FUNCTION "Automatico_linea_2" : VOID	// FC 6
NAME : Auto_L2
VERSION : 0.1
BEGIN
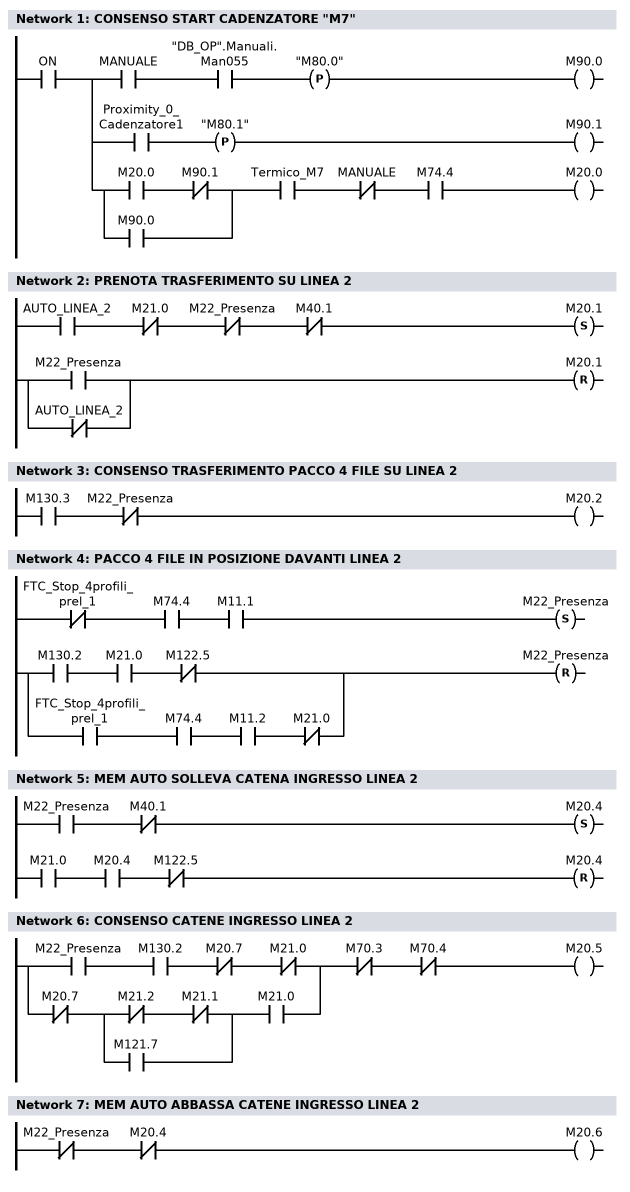
NETWORK
TITLE = CONSENSO START CADENZATORE "M7"
      A     "ON";
      =     L 0.0;
      A     L 0.0;
      A     "MANUALE";
      A     "DB_OP".Manuali.Man055;
      FP    "M80.0";
      =     "M90.0";
      A     L 0.0;
      A     "Proximity_0_Cadenzatore1";
      FP    "M80.1";
      =     "M90.1";
      A     L 0.0;
      A(;
      A     "M20.0";
      AN    "M90.1";
      O     "M90.0";
      );
      A     "Termico_M7";
      AN    "MANUALE";
      A     "M74.4";
      =     "M20.0";
NETWORK
TITLE = PRENOTA TRASFERIMENTO SU LINEA 2
      A     "AUTO_LINEA_2";
      AN    "M21.0";
      AN    "M22_Presenza";
      AN    "M40.1";
      S     "M20.1";
      A(;
      O     "M22_Presenza";
      ON    "AUTO_LINEA_2";
      );
      R     "M20.1";
      NOP   0;
NETWORK
TITLE = CONSENSO TRASFERIMENTO PACCO 4 FILE SU LINEA 2
      A     "M130.3";
      AN    "M22_Presenza";
      =     "M20.2";
NETWORK
TITLE = PACCO 4 FILE IN POSIZIONE DAVANTI LINEA 2
      AN    "FTC_Stop_4profili_prel_1";
      A     "M74.4";
      A     "M11.1";
      S     "M22_Presenza";
      A(;
      A     "M130.2";
      A     "M21.0";
      AN    "M122.5";
      O;
      A     "FTC_Stop_4profili_prel_1";
      A     "M74.4";
      A     "M11.2";
      AN    "M21.0";
      );
      R     "M22_Presenza";
      NOP   0;
NETWORK
TITLE = MEM AUTO SOLLEVA CATENA INGRESSO LINEA 2
      A     "M22_Presenza";
      AN    "M40.1";
      S     "M20.4";
      A     "M21.0";
      A     "M20.4";
      AN    "M122.5";
      R     "M20.4";
      NOP   0;
NETWORK
TITLE = CONSENSO CATENE INGRESSO LINEA 2
      A(;
      A     "M22_Presenza";
      A     "M130.2";
      AN    "M20.7";
      AN    "M21.0";
      O;
      AN    "M20.7";
      A(;
      AN    "M21.2";
      AN    "M21.1";
      O     "M121.7";
      );
      A     "M21.0";
      );
      AN    "M70.3";
      AN    "M70.4";
      =     "M20.5";
NETWORK
TITLE = MEM AUTO ABBASSA CATENE INGRESSO LINEA 2
      AN    "M22_Presenza";
      AN    "M20.4";
      =     "M20.6";
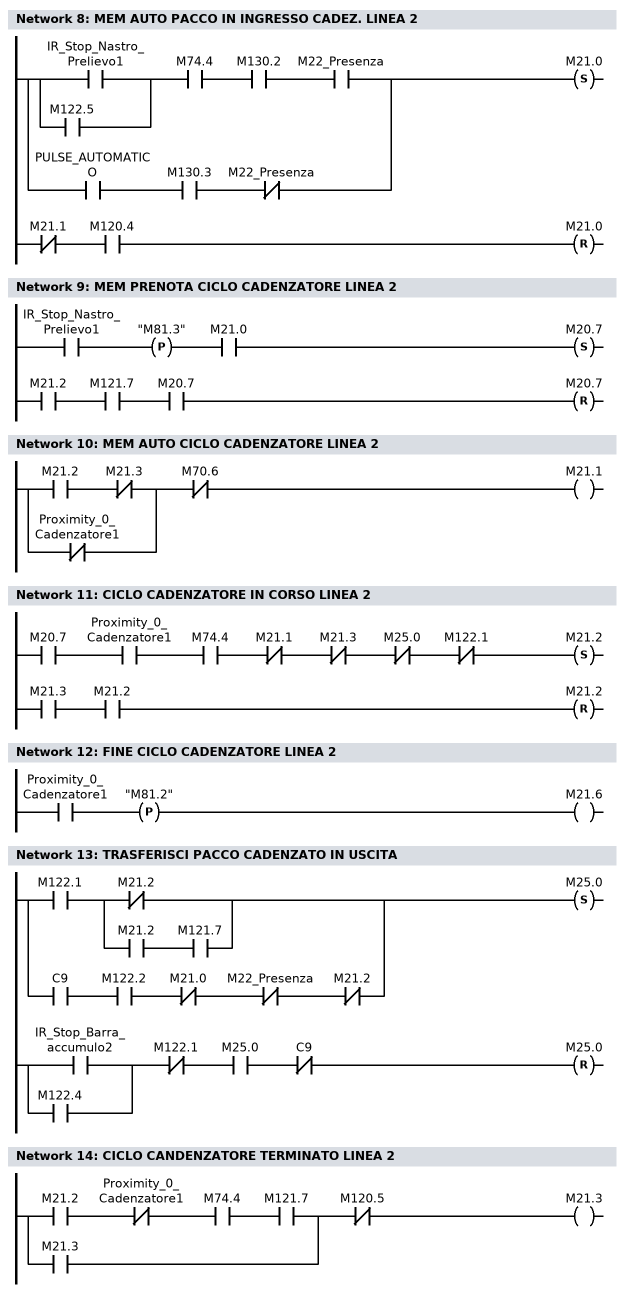
NETWORK
TITLE = MEM AUTO PACCO IN INGRESSO CADEZ. LINEA 2
      A(;
      A(;
      O     "IR_Stop_Nastro_Prelievo1";
      O     "M122.5";
      );
      A     "M74.4";
      A     "M130.2";
      A     "M22_Presenza";
      O;
      A     "PULSE_AUTOMATICO";
      A     "M130.3";
      AN    "M22_Presenza";
      );
      S     "M21.0";
      AN    "M21.1";
      A     "M120.4";
      R     "M21.0";
      NOP   0;
NETWORK
TITLE = MEM PRENOTA CICLO CADENZATORE LINEA 2
      A     "IR_Stop_Nastro_Prelievo1";
      FP    "M81.3";
      A     "M21.0";
      S     "M20.7";
      A     "M21.2";
      A     "M121.7";
      A     "M20.7";
      R     "M20.7";
      NOP   0;
NETWORK
TITLE = MEM AUTO CICLO CADENZATORE LINEA 2
      A(;
      A     "M21.2";
      AN    "M21.3";
      ON    "Proximity_0_Cadenzatore1";
      );
      AN    "M70.6";
      =     "M21.1";
NETWORK
TITLE = CICLO CADENZATORE IN CORSO LINEA 2
      A     "M20.7";
      A     "Proximity_0_Cadenzatore1";
      A     "M74.4";
      AN    "M21.1";
      AN    "M21.3";
      AN    "M25.0";
      AN    "M122.1";
      S     "M21.2";
      A     "M21.3";
      A     "M21.2";
      R     "M21.2";
      NOP   0;
NETWORK
TITLE = FINE CICLO CADENZATORE LINEA 2
      A     "Proximity_0_Cadenzatore1";
      FP    "M81.2";
      =     "M21.6";
NETWORK
TITLE = TRASFERISCI PACCO CADENZATO IN USCITA
      A(;
      A     "M122.1";
      A(;
      ON    "M21.2";
      O;
      A     "M21.2";
      A     "M121.7";
      );
      O;
      A     "C9";
      A     "M122.2";
      AN    "M21.0";
      AN    "M22_Presenza";
      AN    "M21.2";
      );
      S     "M25.0";
      A(;
      O     "IR_Stop_Barra_accumulo2";
      O     "M122.4";
      );
      AN    "M122.1";
      A     "M25.0";
      AN    "C9";
      R     "M25.0";
      NOP   0;
NETWORK
TITLE = CICLO CANDENZATORE TERMINATO LINEA 2
      A(;
      A     "M21.2";
      AN    "Proximity_0_Cadenzatore1";
      A     "M74.4";
      A     "M121.7";
      O     "M21.3";
      );
      AN    "M120.5";
      =     "M21.3";
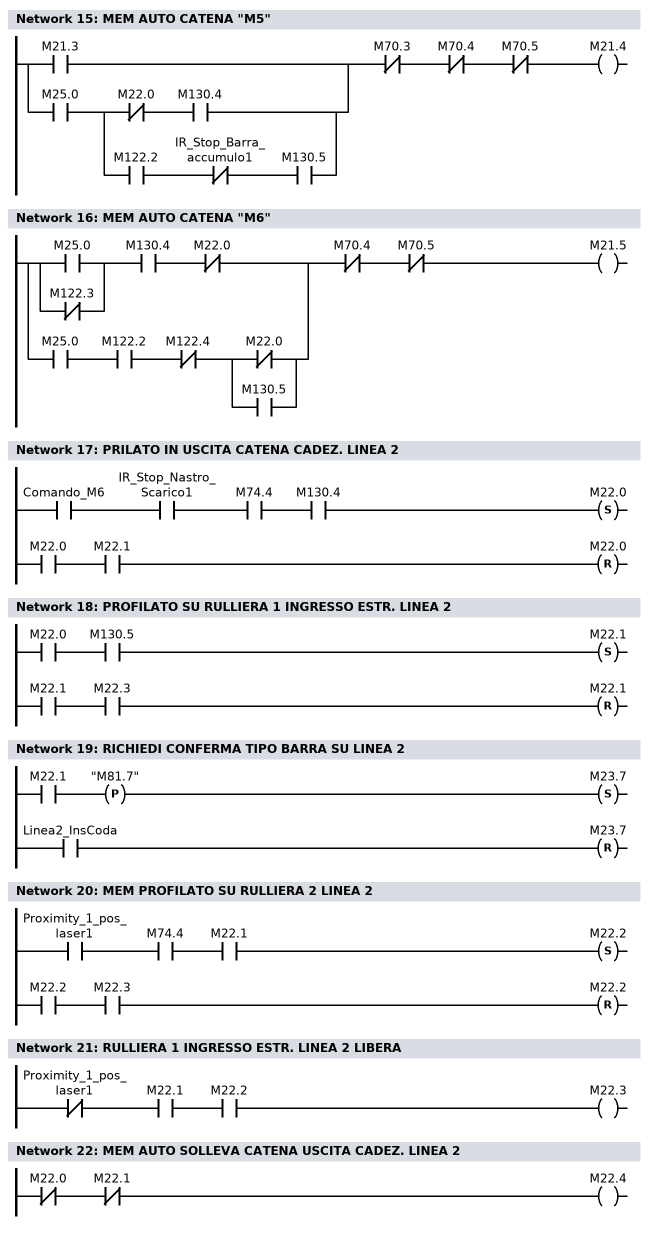
NETWORK
TITLE = MEM AUTO CATENA "M5"
      A(;
      O     "M21.3";
      O;
      A     "M25.0";
      A(;
      AN    "M22.0";
      A     "M130.4";
      O;
      A     "M122.2";
      AN    "IR_Stop_Barra_accumulo1";
      A     "M130.5";
      );
      );
      AN    "M70.3";
      AN    "M70.4";
      AN    "M70.5";
      =     "M21.4";
NETWORK
TITLE = MEM AUTO CATENA "M6"
      A(;
      A(;
      O     "M25.0";
      ON    "M122.3";
      );
      A     "M130.4";
      AN    "M22.0";
      O;
      A     "M25.0";
      A     "M122.2";
      AN    "M122.4";
      A(;
      ON    "M22.0";
      O     "M130.5";
      );
      );
      AN    "M70.4";
      AN    "M70.5";
      =     "M21.5";
NETWORK
TITLE = PRILATO IN USCITA CATENA CADEZ. LINEA 2
      A     "Comando_M6";
      A     "IR_Stop_Nastro_Scarico1";
      A     "M74.4";
      A     "M130.4";
      S     "M22.0";
      A     "M22.0";
      A     "M22.1";
      R     "M22.0";
      NOP   0;
NETWORK
TITLE = PROFILATO SU RULLIERA 1 INGRESSO ESTR. LINEA 2
      A     "M22.0";
      A     "M130.5";
      S     "M22.1";
      A     "M22.1";
      A     "M22.3";
      R     "M22.1";
      NOP   0;
NETWORK
TITLE = RICHIEDI CONFERMA TIPO BARRA SU LINEA 2
      A     "M22.1";
      FP    "M81.7";
      S     "M23.7";
      A     "Linea2_InsCoda";
      R     "M23.7";
      NOP   0;
NETWORK
TITLE = MEM PROFILATO SU RULLIERA 2 LINEA 2
      A     "Proximity_1_pos_laser1";
      A     "M74.4";
      A     "M22.1";
      S     "M22.2";
      A     "M22.2";
      A     "M22.3";
      R     "M22.2";
      NOP   0;
NETWORK
TITLE = RULLIERA 1 INGRESSO ESTR. LINEA 2 LIBERA
      AN    "Proximity_1_pos_laser1";
      A     "M22.1";
      A     "M22.2";
      =     "M22.3";
NETWORK
TITLE = MEM AUTO SOLLEVA CATENA USCITA CADEZ. LINEA 2
      AN    "M22.0";
      AN    "M22.1";
      =     "M22.4";
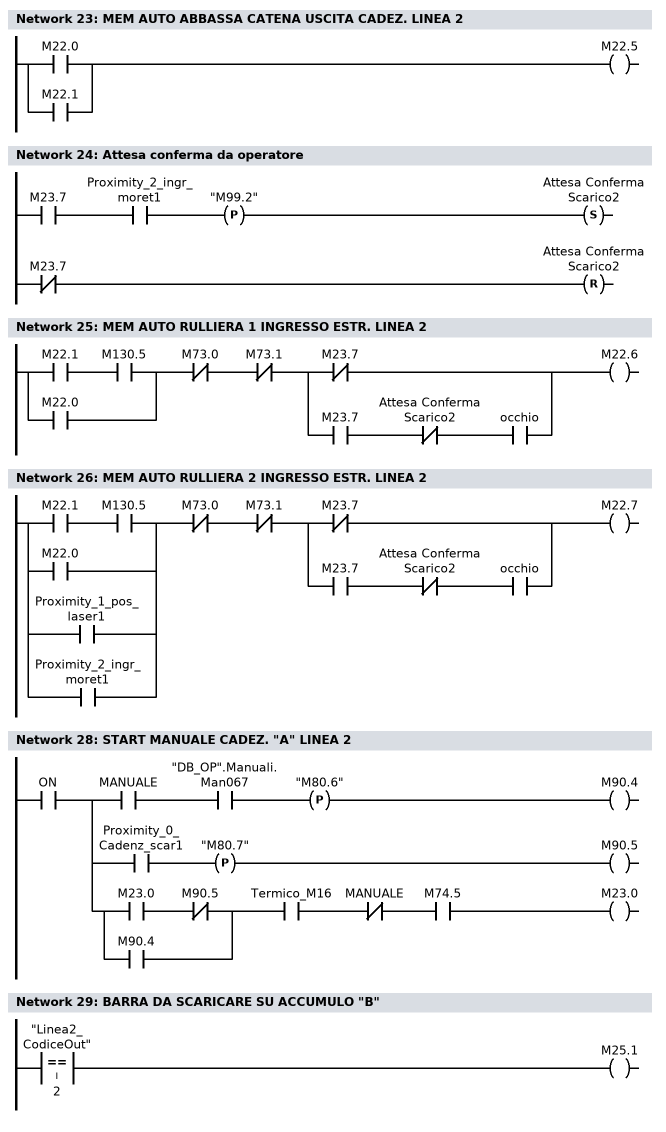
NETWORK
TITLE = MEM AUTO ABBASSA CATENA USCITA CADEZ. LINEA 2
      O     "M22.0";
      O     "M22.1";
      =     "M22.5";
NETWORK
TITLE = Attesa conferma da operatore
      A     "M23.7";
      A     "Proximity_2_ingr_moret1";
      FP    "M99.2";
      S     "Attesa Conferma Scarico2";
      AN    "M23.7";
      R     "Attesa Conferma Scarico2";
      NOP   0;
NETWORK
TITLE = MEM AUTO RULLIERA 1 INGRESSO ESTR. LINEA 2
      A(;
      A     "M22.1";
      A     "M130.5";
      O     "M22.0";
      );
      AN    "M73.0";
      AN    "M73.1";
      A(;
      ON    "M23.7";
      O;
      A     "M23.7";
      AN    "Attesa Conferma Scarico2";
      A     "occhio";
      );
      =     "M22.6";
NETWORK
TITLE = MEM AUTO RULLIERA 2 INGRESSO ESTR. LINEA 2
      A(;
      A     "M22.1";
      A     "M130.5";
      O     "M22.0";
      O     "Proximity_1_pos_laser1";
      O     "Proximity_2_ingr_moret1";
      );
      AN    "M73.0";
      AN    "M73.1";
      A(;
      ON    "M23.7";
      O;
      A     "M23.7";
      AN    "Attesa Conferma Scarico2";
      A     "occhio";
      );
      =     "M22.7";
NETWORK
TITLE =
NETWORK
TITLE = START MANUALE CADEZ. "A" LINEA 2
      A     "ON";
      =     L 0.0;
      A     L 0.0;
      A     "MANUALE";
      A     "DB_OP".Manuali.Man067;
      FP    "M80.6";
      =     "M90.4";
      A     L 0.0;
      A     "Proximity_0_Cadenz_scar1";
      FP    "M80.7";
      =     "M90.5";
      A     L 0.0;
      A(;
      A     "M23.0";
      AN    "M90.5";
      O     "M90.4";
      );
      A     "Termico_M16";
      AN    "MANUALE";
      A     "M74.5";
      =     "M23.0";
NETWORK
TITLE = BARRA DA SCARICARE SU ACCUMULO "B"
      L     "Linea2_CodiceOut";
      L     2;
      ==I;
      =     "M25.1";
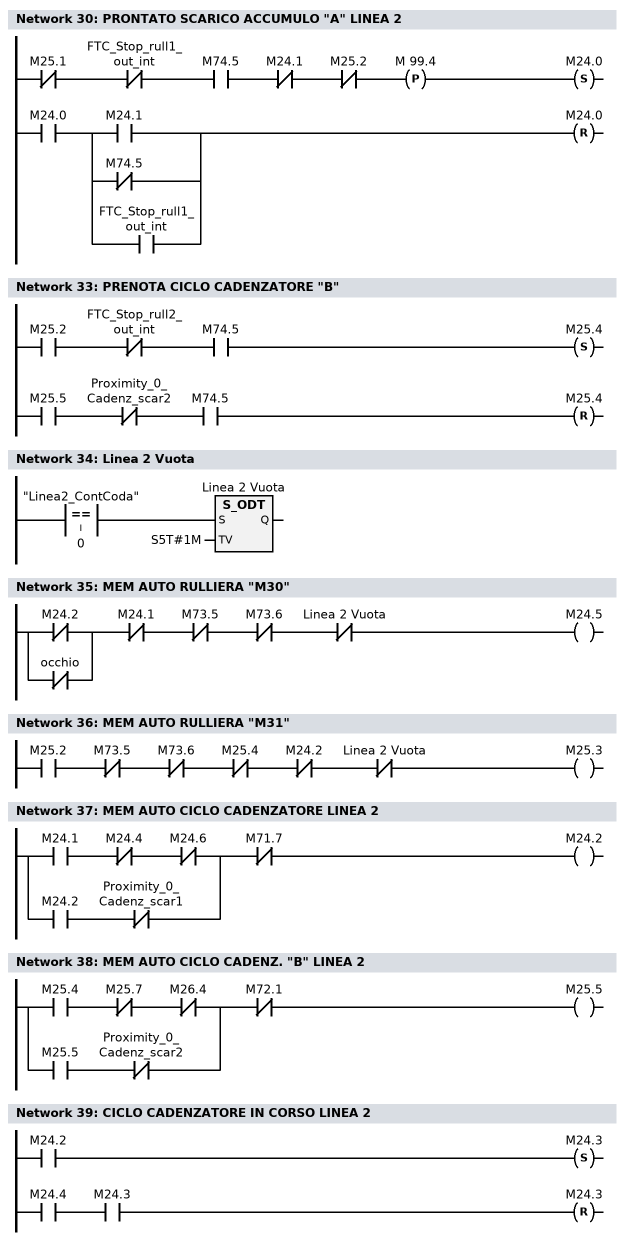
NETWORK
TITLE = PRONTATO SCARICO ACCUMULO "A" LINEA 2
      AN    "M25.1";
      AN    "FTC_Stop_rull1_out_int";
      A     "M74.5";
      AN    "M24.1";
      AN    "M25.2";
      FP    M 99.4;
      S     "M24.0";
      A     "M24.0";
      A(;
      O     "M24.1";
      ON    "M74.5";
      O     "FTC_Stop_rull1_out_int";
      );
      R     "M24.0";
      NOP   0;
NETWORK
TITLE = SPOSTA BASSA RU RULLIERA "M31"
      A(;
      A     "M25.1";
      AN    "FTC_Stop_rull1_out_int";
      A     "M74.5";
      AN    "M24.1";
      S     "M25.2";
      A(;
      A     "M25.4";
      A     "occhio";
      O     "M25.7";
      );
      A     "M25.2";
      R     "M25.2";
      A     "M25.2";
      );
      FP    "M82.1";
      S     "Linea2_DelCoda";
NETWORK
TITLE = PROFILATO PRONTO SU CADEZ. "A" LINEA 2
      A(;
      A(;
      AN    "FTC_Stop_rull1_out_int";
      L     S5T#100MS;
      SD    "T124";
      NOP   0;
      NOP   0;
      NOP   0;
      A     "T124";
      );
      A     "M24.0";
      A     "M74.5";
      S     "M24.1";
      A     "M24.2";
      AN    "Proximity_0_Cadenz_scar1";
      A     "M74.5";
      R     "M24.1";
      A     "M24.1";
      );
      FP    "M82.0";
      S     "Linea2_DelCoda";
NETWORK
TITLE = PRENOTA CICLO CADENZATORE "B"
      A     "M25.2";
      AN    "FTC_Stop_rull2_out_int";
      A     "M74.5";
      S     "M25.4";
      A     "M25.5";
      AN    "Proximity_0_Cadenz_scar2";
      A     "M74.5";
      R     "M25.4";
      NOP   0;
NETWORK
TITLE = Linea 2 Vuota
      A(;
      L     "Linea2_ContCoda";
      L     0;
      ==I;
      );
      L     S5T#1M;
      SD    "Linea 2 Vuota";
      NOP   0;
      NOP   0;
      NOP   0;
      NOP   0;
NETWORK
TITLE = MEM AUTO RULLIERA "M30"
      A(;
      ON    "M24.2";
      ON    "occhio";
      );
      AN    "M24.1";
      AN    "M73.5";
      AN    "M73.6";
      AN    "Linea 2 Vuota";
      =     "M24.5";
NETWORK
TITLE = MEM AUTO RULLIERA "M31"
      A     "M25.2";
      AN    "M73.5";
      AN    "M73.6";
      AN    "M25.4";
      AN    "M24.2";
      AN    "Linea 2 Vuota";
      =     "M25.3";
NETWORK
TITLE = MEM AUTO CICLO CADENZATORE LINEA 2
      A(;
      A     "M24.1";
      AN    "M24.4";
      AN    "M24.6";
      O;
      A     "M24.2";
      AN    "Proximity_0_Cadenz_scar1";
      );
      AN    "M71.7";
      =     "M24.2";
NETWORK
TITLE = MEM AUTO CICLO CADENZ. "B" LINEA 2
      A(;
      A     "M25.4";
      AN    "M25.7";
      AN    "M26.4";
      O;
      A     "M25.5";
      AN    "Proximity_0_Cadenz_scar2";
      );
      AN    "M72.1";
      =     "M25.5";
NETWORK
TITLE = CICLO CADENZATORE IN CORSO LINEA 2
      A     "M24.2";
      S     "M24.3";
      A     "M24.4";
      A     "M24.3";
      R     "M24.3";
      NOP   0;
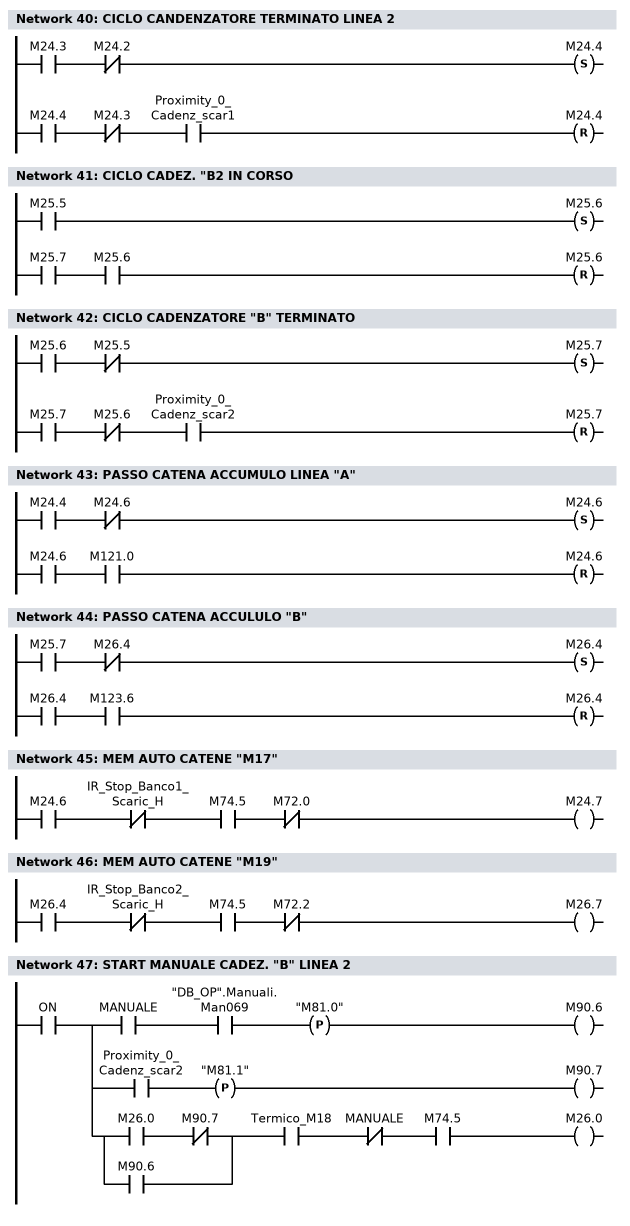
NETWORK
TITLE = CICLO CANDENZATORE TERMINATO LINEA 2
      A     "M24.3";
      AN    "M24.2";
      S     "M24.4";
      A     "M24.4";
      AN    "M24.3";
      A     "Proximity_0_Cadenz_scar1";
      R     "M24.4";
      NOP   0;
NETWORK
TITLE = CICLO CADEZ. "B2 IN CORSO
      A     "M25.5";
      S     "M25.6";
      A     "M25.7";
      A     "M25.6";
      R     "M25.6";
      NOP   0;
NETWORK
TITLE = CICLO CADENZATORE "B" TERMINATO
      A     "M25.6";
      AN    "M25.5";
      S     "M25.7";
      A     "M25.7";
      AN    "M25.6";
      A     "Proximity_0_Cadenz_scar2";
      R     "M25.7";
      NOP   0;
NETWORK
TITLE = PASSO CATENA ACCUMULO LINEA "A"
      A     "M24.4";
      AN    "M24.6";
      S     "M24.6";
      A     "M24.6";
      A     "M121.0";
      R     "M24.6";
      NOP   0;
NETWORK
TITLE = PASSO CATENA ACCULULO "B"
      A     "M25.7";
      AN    "M26.4";
      S     "M26.4";
      A     "M26.4";
      A     "M123.6";
      R     "M26.4";
      NOP   0;
NETWORK
TITLE = MEM AUTO CATENE "M17"
      A     "M24.6";
      AN    "IR_Stop_Banco1_Scaric_H";
      A     "M74.5";
      AN    "M72.0";
      =     "M24.7";
NETWORK
TITLE = MEM AUTO CATENE "M19"
      A     "M26.4";
      AN    "IR_Stop_Banco2_Scaric_H";
      A     "M74.5";
      AN    "M72.2";
      =     "M26.7";
NETWORK
TITLE = START MANUALE CADEZ. "B" LINEA 2
      A     "ON";
      =     L 0.0;
      A     L 0.0;
      A     "MANUALE";
      A     "DB_OP".Manuali.Man069;
      FP    "M81.0";
      =     "M90.6";
      A     L 0.0;
      A     "Proximity_0_Cadenz_scar2";
      FP    "M81.1";
      =     "M90.7";
      A     L 0.0;
      A(;
      A     "M26.0";
      AN    "M90.7";
      O     "M90.6";
      );
      A     "Termico_M18";
      AN    "MANUALE";
      A     "M74.5";
      =     "M26.0";
END_FUNCTION

FUNCTION "PROFIBUS_MM4" : VOID	// FC 10
AUTHOR : PROTEKNO
NAME : MM4
VERSION : 0.1
VAR_INPUT
  Periferic_Address : INT ;
  Drive_On_Off : BOOL ;
  Drive_Reversing : BOOL ;
  Drive_Fault_ACKN : BOOL ;
  Drive_F_Setpoint : REAL ;
END_VAR
VAR_OUTPUT
  Drive_in_operation : BOOL ;
  Drive_Fault_Active : BOOL ;
  Drive_Alarm_Active : BOOL ;
  Freno : BOOL ;
  Drive_F_Act : REAL ;
END_VAR
VAR_TEMP
  Address_E_A : DWORD ;
  SEND : STRUCT
   CW1 : UDT 1;
   f_setpoint : WORD ;
  END_STRUCT ;
  REC : STRUCT
   SW1 : UDT 2;
   f_act : WORD ;
  END_STRUCT ;
END_VAR
BEGIN
NETWORK
TITLE = Trasferimento indirizzo blocco;
      L     #Periferic_Address;
      SLD   3;
      T     #Address_E_A;
NETWORK
TITLE = Status word PZD MM4;
      L     PID [#Address_E_A];
      T     #REC;	//Status word MM4;
NETWORK
TITLE = control bit`s + setpoint
// ---------------------------------------
// IN-Variablen FC
// --------------------------------------
// PZD1 - Steuerwort 1                  // set single bit in the control word 1
      SET;	// set VKE=1
      =     #SEND.CW1.Bit_1;
      =     #SEND.CW1.Bit_2;
      =     #SEND.CW1.Bit_3;
      =     #SEND.CW1.Bit_4;
      =     #SEND.CW1.Bit_5;
      =     #SEND.CW1.Bit_6;
      =     #SEND.CW1.Bit_10;	// setpoint valid
      CLR;	// set VKE=0
      =     #SEND.CW1.Bit_8;
      =     #SEND.CW1.Bit_9;
      =     #SEND.CW1.Bit_12;
      =     #SEND.CW1.Bit_13;
      =     #SEND.CW1.Bit_14;
      =     #SEND.CW1.Bit_15;
      A     #Drive_On_Off;	// on / off ?
      =     #SEND.CW1.Bit_0;
      A     #Drive_Reversing;	// cw / cww ?
      =     #SEND.CW1.Bit_11;
      A     #Drive_Fault_ACKN;	// fault ackn.?
      =     #SEND.CW1.Bit_7;
//  
// PZD2 - Drehzahlsollwert
// gültiger Drehzahlsollwert zwischen 0.00-50 Hz
      L     #Drive_F_Setpoint;	// setpoint [Hz]
      L     0.000000e+00;
      <R;	// setpoinz >0Hz
      JC    N004;
      L     #Drive_F_Setpoint;
      L     7.500000e+01;
      >R;	// setpoint < 75Hz ?
      JC    N004;
      L     #Drive_F_Setpoint;
      L     1.000000e+02;	// 2-Nachkommastellen retten
      *R;
      RND;	//conversion of a 32-bit IEEE floating-point number to 32-bit integer
      L     24576;	// 16384 = 4000HEX = 50Hz
      *D;
      L     7500;
      /D;
      T     #SEND.f_setpoint;
N004: NOP   0;
NETWORK
TITLE = stateword + actual frequency 
// -------------------------------------
// OUT-Variablen FC                     
// -------------------------------------
// PZD 1 - Zustandswort
      A     #REC.SW1.Bit_2;
      =     #Drive_in_operation;
      A     #REC.SW1.Bit_3;
      =     #Drive_Fault_Active;
      A     #REC.SW1.Bit_7;
      =     #Drive_Alarm_Active;
      A     #REC.SW1.Bit_12;
      =     #Freno;
// PZD 2 - Drehzahlistwert
      L     #REC.f_act;
      ITD;
      DTR;
      L     5.000000e+01;	//16383= 4000HEX = 50Hz
      *R;
      L     1.638400e+04;
      /R;
      L     1.000000e+02;
      *R;
      TRUNC;
      ITD;
      DTR;
      L     1.000000e+02;
      /R;
      T     #Drive_F_Act;
NETWORK
TITLE = Control word PZD MM4;
      L     #SEND;	//Control word MM4;
      T     PQD [#Address_E_A];
      BE;
END_FUNCTION

FUNCTION "Comandi_zona_ingresso" : VOID	// FC 14
VERSION : 0.1
BEGIN
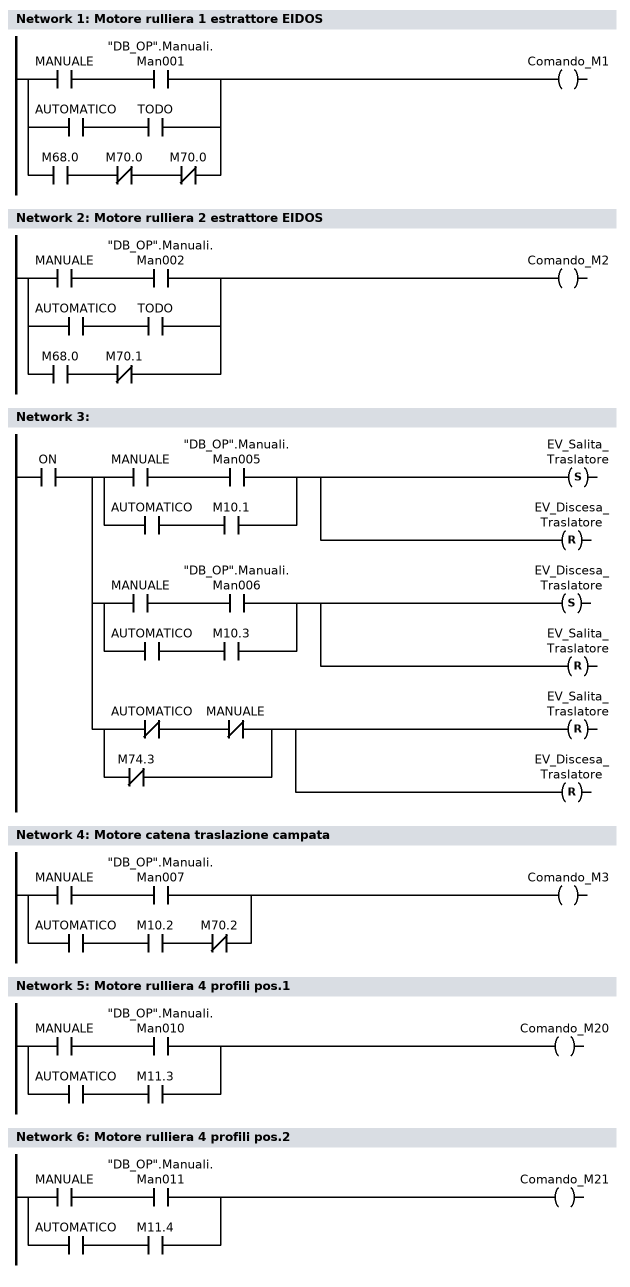
NETWORK
TITLE = Motore rulliera 1 estrattore EIDOS
      A     "MANUALE";
      A     "DB_OP".Manuali.Man001;
      O;
      A     "AUTOMATICO";
      A     "TODO";
      O;
      A     "M68.0";
      AN    "M70.0";
      AN    "M70.0";
      =     "Comando_M1";
NETWORK
TITLE = Motore rulliera 2 estrattore EIDOS
      A     "MANUALE";
      A     "DB_OP".Manuali.Man002;
      O;
      A     "AUTOMATICO";
      A     "TODO";
      O;
      A     "M68.0";
      AN    "M70.1";
      =     "Comando_M2";
NETWORK
TITLE =
      A     "ON";
      =     L 0.0;
      A     L 0.0;
      A(;
      A     "MANUALE";
      A     "DB_OP".Manuali.Man005;
      O;
      A     "AUTOMATICO";
      A     "M10.1";
      );
      S     "EV_Salita_Traslatore";
      R     "EV_Discesa_Traslatore";
      A     L 0.0;
      A(;
      A     "MANUALE";
      A     "DB_OP".Manuali.Man006;
      O;
      A     "AUTOMATICO";
      A     "M10.3";
      );
      S     "EV_Discesa_Traslatore";
      R     "EV_Salita_Traslatore";
      A     L 0.0;
      A(;
      AN    "AUTOMATICO";
      AN    "MANUALE";
      ON    "M74.3";
      );
      R     "EV_Salita_Traslatore";
      R     "EV_Discesa_Traslatore";
NETWORK
TITLE = Motore catena traslazione campata
      A     "MANUALE";
      A     "DB_OP".Manuali.Man007;
      O;
      A     "AUTOMATICO";
      A     "M10.2";
      AN    "M70.2";
      =     "Comando_M3";
NETWORK
TITLE = Motore rulliera 4 profili pos.1
      A     "MANUALE";
      A     "DB_OP".Manuali.Man010;
      O;
      A     "AUTOMATICO";
      A     "M11.3";
      =     "Comando_M20";
NETWORK
TITLE = Motore rulliera 4 profili pos.2
      A     "MANUALE";
      A     "DB_OP".Manuali.Man011;
      O;
      A     "AUTOMATICO";
      A     "M11.4";
      =     "Comando_M21";
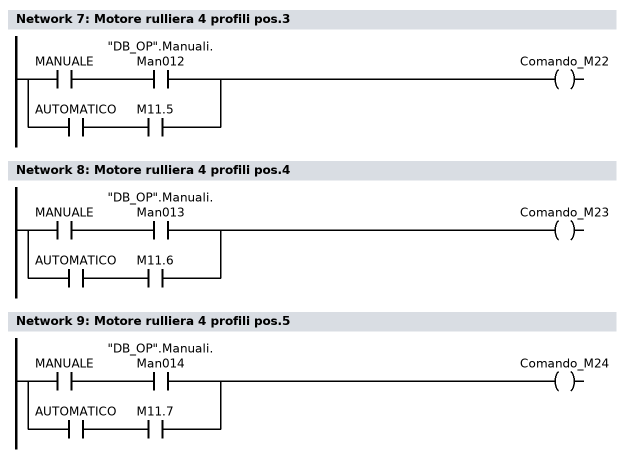
NETWORK
TITLE = Motore rulliera 4 profili pos.3
      A     "MANUALE";
      A     "DB_OP".Manuali.Man012;
      O;
      A     "AUTOMATICO";
      A     "M11.5";
      =     "Comando_M22";
NETWORK
TITLE = Motore rulliera 4 profili pos.4
      A     "MANUALE";
      A     "DB_OP".Manuali.Man013;
      O;
      A     "AUTOMATICO";
      A     "M11.6";
      =     "Comando_M23";
NETWORK
TITLE = Motore rulliera 4 profili pos.5
      A     "MANUALE";
      A     "DB_OP".Manuali.Man014;
      O;
      A     "AUTOMATICO";
      A     "M11.7";
      =     "Comando_M24";
END_FUNCTION

FUNCTION "Comandi_linea_1" : VOID	// FC 15
VERSION : 0.1
BEGIN
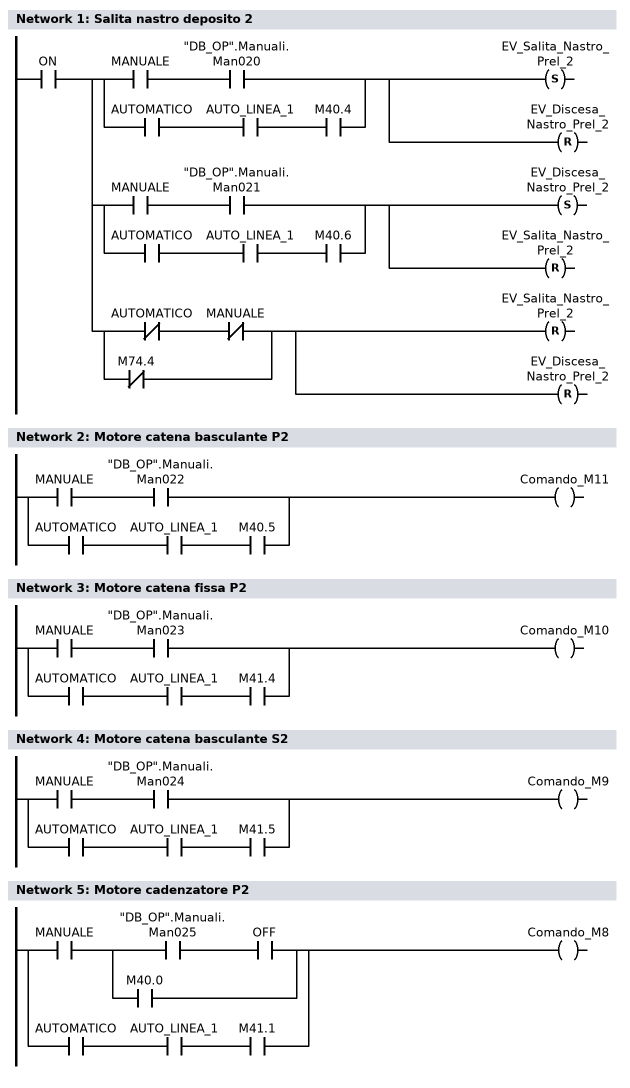
NETWORK
TITLE = Salita nastro deposito 2
      A     "ON";
      =     L 0.0;
      A     L 0.0;
      A(;
      A     "MANUALE";
      A     "DB_OP".Manuali.Man020;
      O;
      A     "AUTOMATICO";
      A     "AUTO_LINEA_1";
      A     "M40.4";
      );
      S     "EV_Salita_Nastro_Prel_2";
      R     "EV_Discesa_Nastro_Prel_2";
      A     L 0.0;
      A(;
      A     "MANUALE";
      A     "DB_OP".Manuali.Man021;
      O;
      A     "AUTOMATICO";
      A     "AUTO_LINEA_1";
      A     "M40.6";
      );
      S     "EV_Discesa_Nastro_Prel_2";
      R     "EV_Salita_Nastro_Prel_2";
      A     L 0.0;
      A(;
      AN    "AUTOMATICO";
      AN    "MANUALE";
      ON    "M74.4";
      );
      R     "EV_Salita_Nastro_Prel_2";
      R     "EV_Discesa_Nastro_Prel_2";
NETWORK
TITLE = Motore catena basculante P2
      A     "MANUALE";
      A     "DB_OP".Manuali.Man022;
      O;
      A     "AUTOMATICO";
      A     "AUTO_LINEA_1";
      A     "M40.5";
      =     "Comando_M11";
NETWORK
TITLE = Motore catena fissa P2
      A     "MANUALE";
      A     "DB_OP".Manuali.Man023;
      O;
      A     "AUTOMATICO";
      A     "AUTO_LINEA_1";
      A     "M41.4";
      =     "Comando_M10";
NETWORK
TITLE = Motore catena basculante S2
      A     "MANUALE";
      A     "DB_OP".Manuali.Man024;
      O;
      A     "AUTOMATICO";
      A     "AUTO_LINEA_1";
      A     "M41.5";
      =     "Comando_M9";
NETWORK
TITLE = Motore cadenzatore P2
      A     "MANUALE";
      A(;
      A     "DB_OP".Manuali.Man025;
      A     "OFF";
      O     "M40.0";
      );
      O;
      A     "AUTOMATICO";
      A     "AUTO_LINEA_1";
      A     "M41.1";
      =     "Comando_M8";
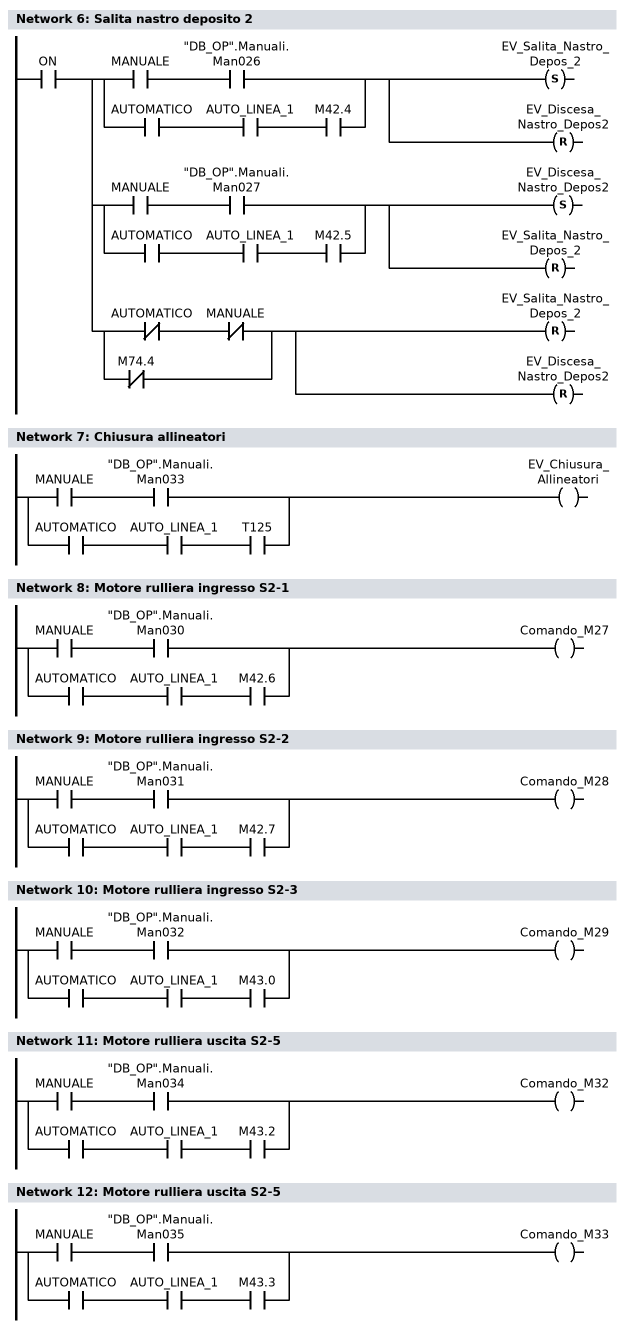
NETWORK
TITLE = Salita nastro deposito 2
      A     "ON";
      =     L 0.0;
      A     L 0.0;
      A(;
      A     "MANUALE";
      A     "DB_OP".Manuali.Man026;
      O;
      A     "AUTOMATICO";
      A     "AUTO_LINEA_1";
      A     "M42.4";
      );
      S     "EV_Salita_Nastro_Depos_2";
      R     "EV_Discesa_Nastro_Depos2";
      A     L 0.0;
      A(;
      A     "MANUALE";
      A     "DB_OP".Manuali.Man027;
      O;
      A     "AUTOMATICO";
      A     "AUTO_LINEA_1";
      A     "M42.5";
      );
      S     "EV_Discesa_Nastro_Depos2";
      R     "EV_Salita_Nastro_Depos_2";
      A     L 0.0;
      A(;
      AN    "AUTOMATICO";
      AN    "MANUALE";
      ON    "M74.4";
      );
      R     "EV_Salita_Nastro_Depos_2";
      R     "EV_Discesa_Nastro_Depos2";
NETWORK
TITLE = Chiusura allineatori
      A     "MANUALE";
      A     "DB_OP".Manuali.Man033;
      O;
      A     "AUTOMATICO";
      A     "AUTO_LINEA_1";
      A     "T125";
      =     "EV_Chiusura_Allineatori";
NETWORK
TITLE = Motore rulliera ingresso S2-1
      A     "MANUALE";
      A     "DB_OP".Manuali.Man030;
      O;
      A     "AUTOMATICO";
      A     "AUTO_LINEA_1";
      A     "M42.6";
      =     "Comando_M27";
NETWORK
TITLE = Motore rulliera ingresso S2-2
      A     "MANUALE";
      A     "DB_OP".Manuali.Man031;
      O;
      A     "AUTOMATICO";
      A     "AUTO_LINEA_1";
      A     "M42.7";
      =     "Comando_M28";
NETWORK
TITLE = Motore rulliera ingresso S2-3
      A     "MANUALE";
      A     "DB_OP".Manuali.Man032;
      O;
      A     "AUTOMATICO";
      A     "AUTO_LINEA_1";
      A     "M43.0";
      =     "Comando_M29";
NETWORK
TITLE = Motore rulliera uscita S2-5
      A     "MANUALE";
      A     "DB_OP".Manuali.Man034;
      O;
      A     "AUTOMATICO";
      A     "AUTO_LINEA_1";
      A     "M43.2";
      =     "Comando_M32";
NETWORK
TITLE = Motore rulliera uscita S2-5
      A     "MANUALE";
      A     "DB_OP".Manuali.Man035;
      O;
      A     "AUTOMATICO";
      A     "AUTO_LINEA_1";
      A     "M43.3";
      =     "Comando_M33";
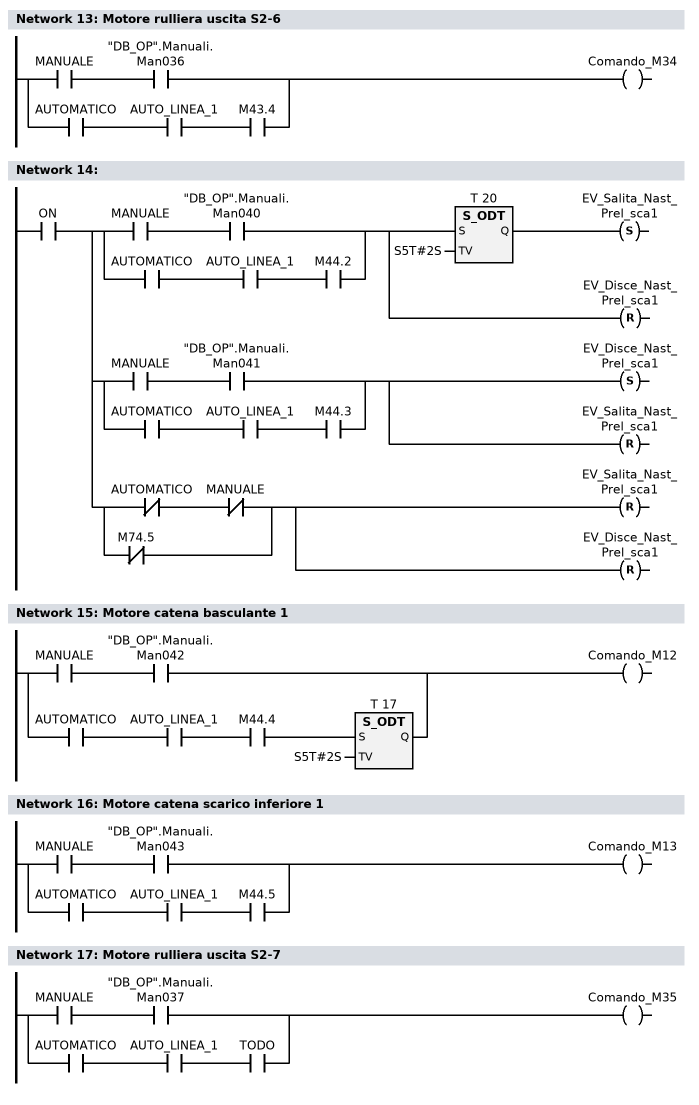
NETWORK
TITLE = Motore rulliera uscita S2-6
      A     "MANUALE";
      A     "DB_OP".Manuali.Man036;
      O;
      A     "AUTOMATICO";
      A     "AUTO_LINEA_1";
      A     "M43.4";
      =     "Comando_M34";
NETWORK
TITLE =
      A     "ON";
      =     L 0.0;
      A     L 0.0;
      A(;
      A     "MANUALE";
      A     "DB_OP".Manuali.Man040;
      O;
      A     "AUTOMATICO";
      A     "AUTO_LINEA_1";
      A     "M44.2";
      );
      =     L 0.1;
      A     L 0.1;
      L     S5T#2S;
      SD    T 20;
      NOP   0;
      NOP   0;
      NOP   0;
      A     T 20;
      S     "EV_Salita_Nast_Prel_sca1";
      A     L 0.1;
      BLD   102;
      R     "EV_Disce_Nast_Prel_sca1";
      A     L 0.0;
      A(;
      A     "MANUALE";
      A     "DB_OP".Manuali.Man041;
      O;
      A     "AUTOMATICO";
      A     "AUTO_LINEA_1";
      A     "M44.3";
      );
      S     "EV_Disce_Nast_Prel_sca1";
      R     "EV_Salita_Nast_Prel_sca1";
      A     L 0.0;
      A(;
      AN    "AUTOMATICO";
      AN    "MANUALE";
      ON    "M74.5";
      );
      R     "EV_Salita_Nast_Prel_sca1";
      R     "EV_Disce_Nast_Prel_sca1";
NETWORK
TITLE = Motore catena basculante 1
      A     "MANUALE";
      A     "DB_OP".Manuali.Man042;
      O(;
      A     "AUTOMATICO";
      A     "AUTO_LINEA_1";
      A     "M44.4";
      L     S5T#2S;
      SD    T 17;
      NOP   0;
      NOP   0;
      NOP   0;
      A     T 17;
      );
      =     "Comando_M12";
NETWORK
TITLE = Motore catena scarico inferiore 1
      A     "MANUALE";
      A     "DB_OP".Manuali.Man043;
      O;
      A     "AUTOMATICO";
      A     "AUTO_LINEA_1";
      A     "M44.5";
      =     "Comando_M13";
NETWORK
TITLE = Motore rulliera uscita S2-7
      A     "MANUALE";
      A     "DB_OP".Manuali.Man037;
      O;
      A     "AUTOMATICO";
      A     "AUTO_LINEA_1";
      A     "TODO";
      =     "Comando_M35";
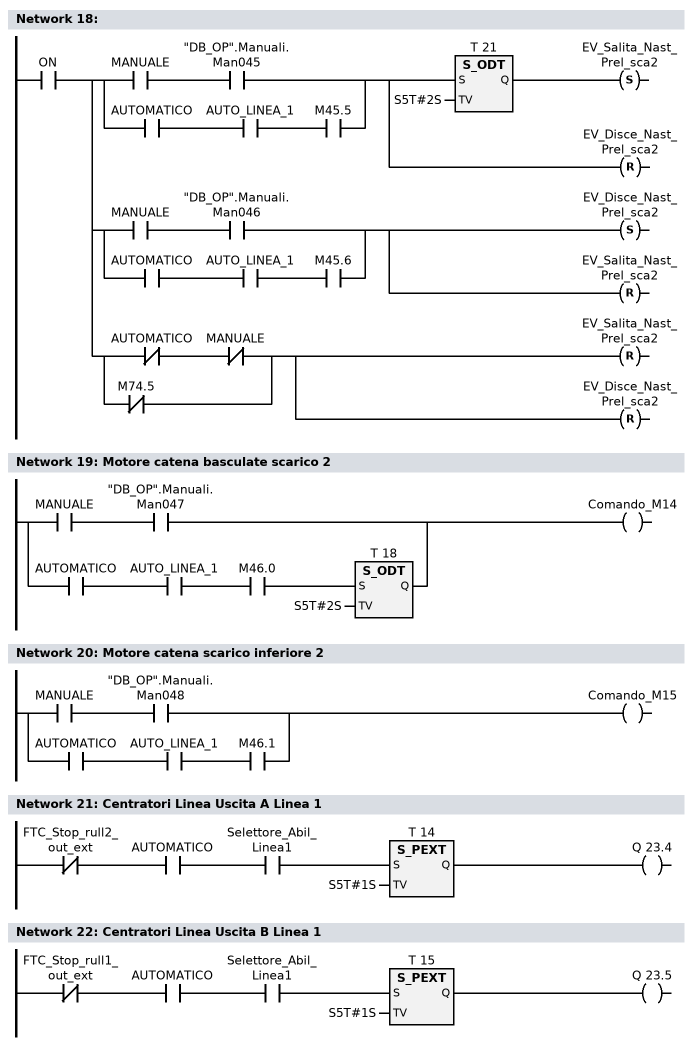
NETWORK
TITLE =
      A     "ON";
      =     L 0.0;
      A     L 0.0;
      A(;
      A     "MANUALE";
      A     "DB_OP".Manuali.Man045;
      O;
      A     "AUTOMATICO";
      A     "AUTO_LINEA_1";
      A     "M45.5";
      );
      =     L 0.1;
      A     L 0.1;
      L     S5T#2S;
      SD    T 21;
      NOP   0;
      NOP   0;
      NOP   0;
      A     T 21;
      S     "EV_Salita_Nast_Prel_sca2";
      A     L 0.1;
      BLD   102;
      R     "EV_Disce_Nast_Prel_sca2";
      A     L 0.0;
      A(;
      A     "MANUALE";
      A     "DB_OP".Manuali.Man046;
      O;
      A     "AUTOMATICO";
      A     "AUTO_LINEA_1";
      A     "M45.6";
      );
      S     "EV_Disce_Nast_Prel_sca2";
      R     "EV_Salita_Nast_Prel_sca2";
      A     L 0.0;
      A(;
      AN    "AUTOMATICO";
      AN    "MANUALE";
      ON    "M74.5";
      );
      R     "EV_Salita_Nast_Prel_sca2";
      R     "EV_Disce_Nast_Prel_sca2";
NETWORK
TITLE = Motore catena basculate scarico 2
      A     "MANUALE";
      A     "DB_OP".Manuali.Man047;
      O(;
      A     "AUTOMATICO";
      A     "AUTO_LINEA_1";
      A     "M46.0";
      L     S5T#2S;
      SD    T 18;
      NOP   0;
      NOP   0;
      NOP   0;
      A     T 18;
      );
      =     "Comando_M14";
NETWORK
TITLE = Motore catena scarico inferiore 2
      A     "MANUALE";
      A     "DB_OP".Manuali.Man048;
      O;
      A     "AUTOMATICO";
      A     "AUTO_LINEA_1";
      A     "M46.1";
      =     "Comando_M15";
NETWORK
TITLE = Centratori Linea Uscita A Linea 1
      AN    "FTC_Stop_rull2_out_ext";
      A     "AUTOMATICO";
      A     "Selettore_Abil_Linea1";
      L     S5T#1S;
      SE    T 14;
      NOP   0;
      NOP   0;
      NOP   0;
      A     T 14;
      =     Q 23.4;
NETWORK
TITLE = Centratori Linea Uscita B Linea 1
      AN    "FTC_Stop_rull1_out_ext";
      A     "AUTOMATICO";
      A     "Selettore_Abil_Linea1";
      L     S5T#1S;
      SE    T 15;
      NOP   0;
      NOP   0;
      NOP   0;
      A     T 15;
      =     Q 23.5;
END_FUNCTION

FUNCTION "Comandi_linea_2" : VOID	// FC 16
VERSION : 0.1
BEGIN
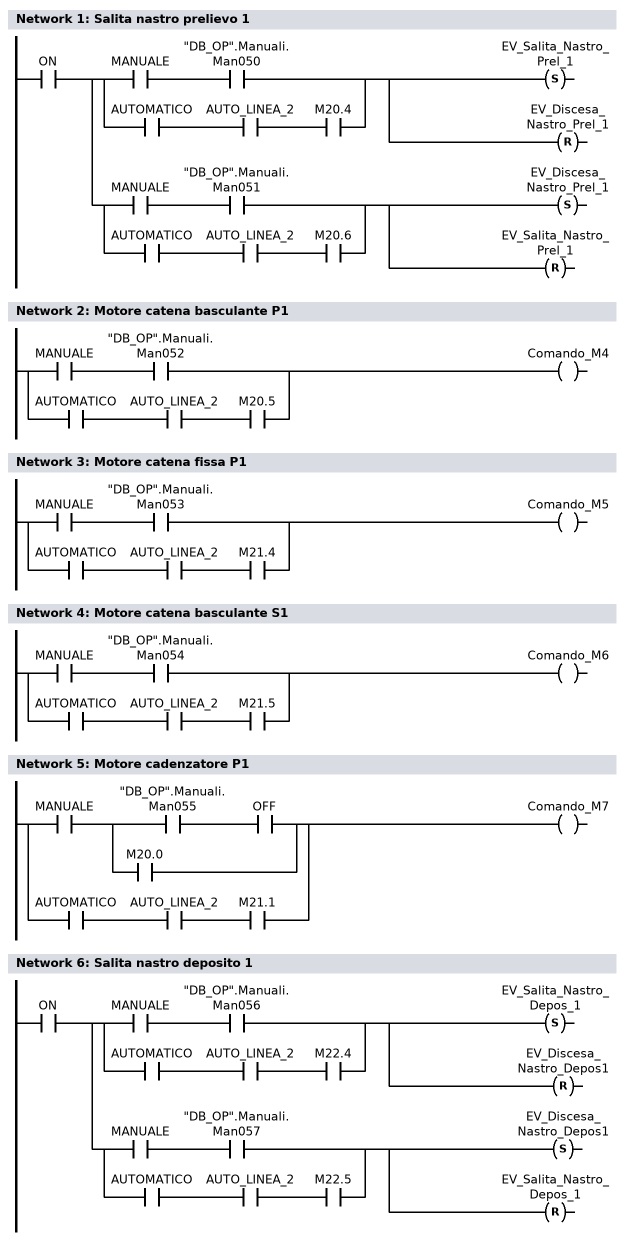
NETWORK
TITLE = Salita nastro prelievo 1
      A     "ON";
      =     L 0.0;
      A     L 0.0;
      A(;
      A     "MANUALE";
      A     "DB_OP".Manuali.Man050;
      O;
      A     "AUTOMATICO";
      A     "AUTO_LINEA_2";
      A     "M20.4";
      );
      S     "EV_Salita_Nastro_Prel_1";
      R     "EV_Discesa_Nastro_Prel_1";
      A     L 0.0;
      A(;
      A     "MANUALE";
      A     "DB_OP".Manuali.Man051;
      O;
      A     "AUTOMATICO";
      A     "AUTO_LINEA_2";
      A     "M20.6";
      );
      S     "EV_Discesa_Nastro_Prel_1";
      R     "EV_Salita_Nastro_Prel_1";
NETWORK
TITLE = Motore catena basculante P1
      A     "MANUALE";
      A     "DB_OP".Manuali.Man052;
      O;
      A     "AUTOMATICO";
      A     "AUTO_LINEA_2";
      A     "M20.5";
      =     "Comando_M4";
NETWORK
TITLE = Motore catena fissa P1
      A     "MANUALE";
      A     "DB_OP".Manuali.Man053;
      O;
      A     "AUTOMATICO";
      A     "AUTO_LINEA_2";
      A     "M21.4";
      =     "Comando_M5";
NETWORK
TITLE = Motore catena basculante S1
      A     "MANUALE";
      A     "DB_OP".Manuali.Man054;
      O;
      A     "AUTOMATICO";
      A     "AUTO_LINEA_2";
      A     "M21.5";
      =     "Comando_M6";
NETWORK
TITLE = Motore cadenzatore P1
      A     "MANUALE";
      A(;
      A     "DB_OP".Manuali.Man055;
      A     "OFF";
      O     "M20.0";
      );
      O;
      A     "AUTOMATICO";
      A     "AUTO_LINEA_2";
      A     "M21.1";
      =     "Comando_M7";
NETWORK
TITLE = Salita nastro deposito 1
      A     "ON";
      =     L 0.0;
      A     L 0.0;
      A(;
      A     "MANUALE";
      A     "DB_OP".Manuali.Man056;
      O;
      A     "AUTOMATICO";
      A     "AUTO_LINEA_2";
      A     "M22.4";
      );
      S     "EV_Salita_Nastro_Depos_1";
      R     "EV_Discesa_Nastro_Depos1";
      A     L 0.0;
      A(;
      A     "MANUALE";
      A     "DB_OP".Manuali.Man057;
      O;
      A     "AUTOMATICO";
      A     "AUTO_LINEA_2";
      A     "M22.5";
      );
      S     "EV_Discesa_Nastro_Depos1";
      R     "EV_Salita_Nastro_Depos_1";
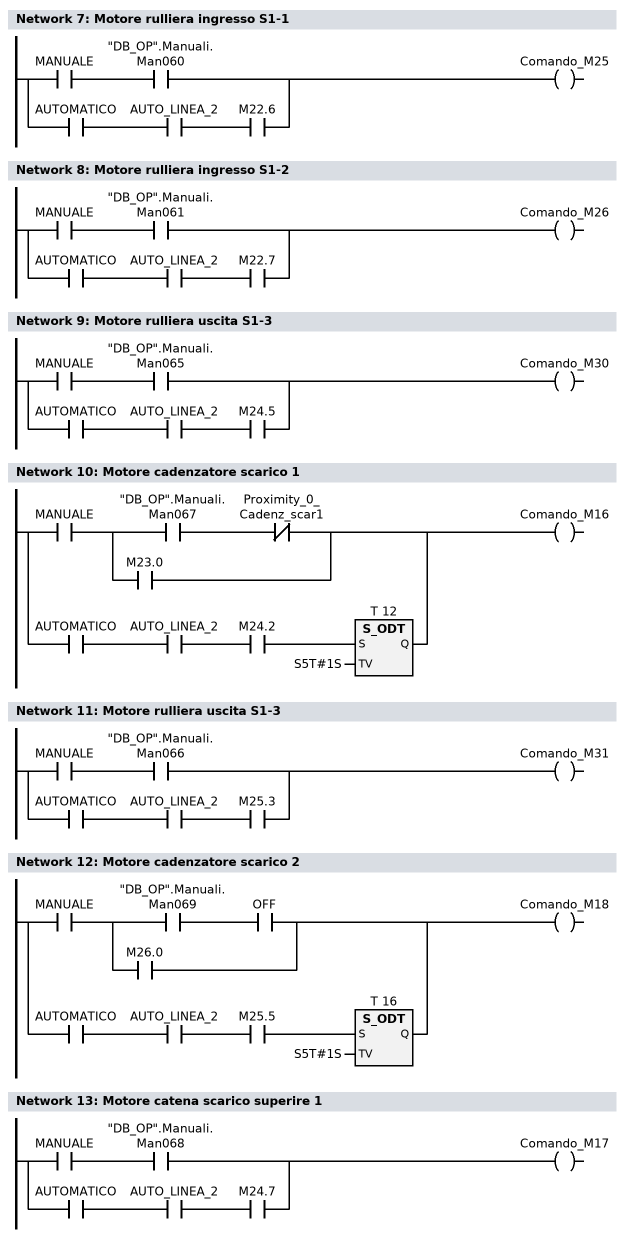
NETWORK
TITLE = Motore rulliera ingresso S1-1
      A     "MANUALE";
      A     "DB_OP".Manuali.Man060;
      O;
      A     "AUTOMATICO";
      A     "AUTO_LINEA_2";
      A     "M22.6";
      =     "Comando_M25";
NETWORK
TITLE = Motore rulliera ingresso S1-2
      A     "MANUALE";
      A     "DB_OP".Manuali.Man061;
      O;
      A     "AUTOMATICO";
      A     "AUTO_LINEA_2";
      A     "M22.7";
      =     "Comando_M26";
NETWORK
TITLE = Motore rulliera uscita S1-3
      A     "MANUALE";
      A     "DB_OP".Manuali.Man065;
      O;
      A     "AUTOMATICO";
      A     "AUTO_LINEA_2";
      A     "M24.5";
      =     "Comando_M30";
NETWORK
TITLE = Motore cadenzatore scarico 1
      A     "MANUALE";
      A(;
      A     "DB_OP".Manuali.Man067;
      AN    "Proximity_0_Cadenz_scar1";
      O     "M23.0";
      );
      O(;
      A     "AUTOMATICO";
      A     "AUTO_LINEA_2";
      A     "M24.2";
      L     S5T#1S;
      SD    T 12;
      NOP   0;
      NOP   0;
      NOP   0;
      A     T 12;
      );
      =     "Comando_M16";
NETWORK
TITLE = Motore rulliera uscita S1-3
      A     "MANUALE";
      A     "DB_OP".Manuali.Man066;
      O;
      A     "AUTOMATICO";
      A     "AUTO_LINEA_2";
      A     "M25.3";
      =     "Comando_M31";
NETWORK
TITLE = Motore cadenzatore scarico 2
      A     "MANUALE";
      A(;
      A     "DB_OP".Manuali.Man069;
      A     "OFF";
      O     "M26.0";
      );
      O(;
      A     "AUTOMATICO";
      A     "AUTO_LINEA_2";
      A     "M25.5";
      L     S5T#1S;
      SD    T 16;
      NOP   0;
      NOP   0;
      NOP   0;
      A     T 16;
      );
      =     "Comando_M18";
NETWORK
TITLE = Motore catena scarico superire 1
      A     "MANUALE";
      A     "DB_OP".Manuali.Man068;
      O;
      A     "AUTOMATICO";
      A     "AUTO_LINEA_2";
      A     "M24.7";
      =     "Comando_M17";
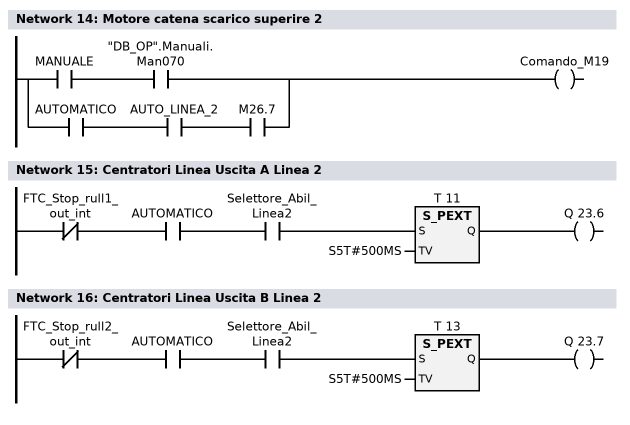
NETWORK
TITLE = Motore catena scarico superire 2
      A     "MANUALE";
      A     "DB_OP".Manuali.Man070;
      O;
      A     "AUTOMATICO";
      A     "AUTO_LINEA_2";
      A     "M26.7";
      =     "Comando_M19";
NETWORK
TITLE = Centratori Linea Uscita A Linea 2
      AN    "FTC_Stop_rull1_out_int";
      A     "AUTOMATICO";
      A     "Selettore_Abil_Linea2";
      L     S5T#500MS;
      SE    T 11;
      NOP   0;
      NOP   0;
      NOP   0;
      A     T 11;
      =     Q 23.6;
NETWORK
TITLE = Centratori Linea Uscita B Linea 2
      AN    "FTC_Stop_rull2_out_int";
      A     "AUTOMATICO";
      A     "Selettore_Abil_Linea2";
      L     S5T#500MS;
      SE    T 13;
      NOP   0;
      NOP   0;
      NOP   0;
      A     T 13;
      =     Q 23.7;
END_FUNCTION

FUNCTION "Comandi_Inverter" : VOID	// FC 17
VERSION : 0.1
VAR_TEMP
  Temp1 : BOOL ;
  Temp2 : BOOL ;
  Temp3 : BOOL ;
  Temp4 : BOOL ;
  RTemp1 : REAL ;
END_VAR
BEGIN
NETWORK
TITLE =
      CALL  "PROFIBUS_MM4" (
           Periferic_Address        := 280,
           Drive_On_Off             := "Comando_M20",
           Drive_Reversing          := FALSE,
           Drive_Fault_ACKN         := FALSE,
           Drive_F_Setpoint         := 7.000000e+01,
           Drive_in_operation       := #Temp1,
           Drive_Fault_Active       := "M66.0",
           Drive_Alarm_Active       := #Temp3,
           Freno                    := #Temp4,
           Drive_F_Act              := #RTemp1);
NETWORK
TITLE =
      CALL  "PROFIBUS_MM4" (
           Periferic_Address        := 292,
           Drive_On_Off             := "Comando_M21",
           Drive_Reversing          := FALSE,
           Drive_Fault_ACKN         := FALSE,
           Drive_F_Setpoint         := 7.000000e+01,
           Drive_in_operation       := #Temp1,
           Drive_Fault_Active       := "M66.1",
           Drive_Alarm_Active       := #Temp3,
           Freno                    := #Temp4,
           Drive_F_Act              := #RTemp1);
NETWORK
TITLE =
      CALL  "PROFIBUS_MM4" (
           Periferic_Address        := 304,
           Drive_On_Off             := "Comando_M22",
           Drive_Reversing          := FALSE,
           Drive_Fault_ACKN         := FALSE,
           Drive_F_Setpoint         := 7.000000e+01,
           Drive_in_operation       := #Temp1,
           Drive_Fault_Active       := "M66.2",
           Drive_Alarm_Active       := #Temp3,
           Freno                    := #Temp4,
           Drive_F_Act              := #RTemp1);
NETWORK
TITLE =
      CALL  "PROFIBUS_MM4" (
           Periferic_Address        := 316,
           Drive_On_Off             := "Comando_M23",
           Drive_Reversing          := FALSE,
           Drive_Fault_ACKN         := FALSE,
           Drive_F_Setpoint         := 7.000000e+01,
           Drive_in_operation       := #Temp1,
           Drive_Fault_Active       := "M66.3",
           Drive_Alarm_Active       := #Temp3,
           Freno                    := #Temp4,
           Drive_F_Act              := #RTemp1);
NETWORK
TITLE =
      CALL  "PROFIBUS_MM4" (
           Periferic_Address        := 328,
           Drive_On_Off             := "Comando_M24",
           Drive_Reversing          := FALSE,
           Drive_Fault_ACKN         := FALSE,
           Drive_F_Setpoint         := 7.000000e+01,
           Drive_in_operation       := #Temp1,
           Drive_Fault_Active       := "M66.4",
           Drive_Alarm_Active       := #Temp3,
           Freno                    := #Temp4,
           Drive_F_Act              := #RTemp1);
NETWORK
TITLE =
      CALL  "PROFIBUS_MM4" (
           Periferic_Address        := 340,
           Drive_On_Off             := "Comando_M25",
           Drive_Reversing          := FALSE,
           Drive_Fault_ACKN         := FALSE,
           Drive_F_Setpoint         := 5.000000e+01,
           Drive_in_operation       := #Temp1,
           Drive_Fault_Active       := "M66.5",
           Drive_Alarm_Active       := #Temp3,
           Freno                    := #Temp4,
           Drive_F_Act              := #RTemp1);
NETWORK
TITLE =
      CALL  "PROFIBUS_MM4" (
           Periferic_Address        := 352,
           Drive_On_Off             := "Comando_M26",
           Drive_Reversing          := FALSE,
           Drive_Fault_ACKN         := FALSE,
           Drive_F_Setpoint         := 5.000000e+01,
           Drive_in_operation       := #Temp1,
           Drive_Fault_Active       := "M66.6",
           Drive_Alarm_Active       := #Temp3,
           Freno                    := #Temp4,
           Drive_F_Act              := #RTemp1);
NETWORK
TITLE =
      CALL  "PROFIBUS_MM4" (
           Periferic_Address        := 364,
           Drive_On_Off             := "Comando_M27",
           Drive_Reversing          := FALSE,
           Drive_Fault_ACKN         := FALSE,
           Drive_F_Setpoint         := 5.000000e+01,
           Drive_in_operation       := #Temp1,
           Drive_Fault_Active       := "M66.7",
           Drive_Alarm_Active       := #Temp3,
           Freno                    := #Temp4,
           Drive_F_Act              := #RTemp1);
NETWORK
TITLE =
      CALL  "PROFIBUS_MM4" (
           Periferic_Address        := 376,
           Drive_On_Off             := "Comando_M28",
           Drive_Reversing          := FALSE,
           Drive_Fault_ACKN         := FALSE,
           Drive_F_Setpoint         := 5.000000e+01,
           Drive_in_operation       := #Temp1,
           Drive_Fault_Active       := "M67.0",
           Drive_Alarm_Active       := #Temp3,
           Freno                    := #Temp4,
           Drive_F_Act              := #RTemp1);
NETWORK
TITLE =
      CALL  "PROFIBUS_MM4" (
           Periferic_Address        := 388,
           Drive_On_Off             := "Comando_M29",
           Drive_Reversing          := FALSE,
           Drive_Fault_ACKN         := FALSE,
           Drive_F_Setpoint         := 5.000000e+01,
           Drive_in_operation       := #Temp1,
           Drive_Fault_Active       := "M67.1",
           Drive_Alarm_Active       := #Temp3,
           Freno                    := #Temp4,
           Drive_F_Act              := #RTemp1);
NETWORK
TITLE =
      CALL  "PROFIBUS_MM4" (
           Periferic_Address        := 400,
           Drive_On_Off             := "Comando_M30",
           Drive_Reversing          := FALSE,
           Drive_Fault_ACKN         := FALSE,
           Drive_F_Setpoint         := 5.000000e+01,
           Drive_in_operation       := #Temp1,
           Drive_Fault_Active       := "M67.2",
           Drive_Alarm_Active       := #Temp3,
           Freno                    := #Temp4,
           Drive_F_Act              := #RTemp1);
NETWORK
TITLE =
      CALL  "PROFIBUS_MM4" (
           Periferic_Address        := 412,
           Drive_On_Off             := "Comando_M31",
           Drive_Reversing          := FALSE,
           Drive_Fault_ACKN         := FALSE,
           Drive_F_Setpoint         := 5.000000e+01,
           Drive_in_operation       := #Temp1,
           Drive_Fault_Active       := "M67.3",
           Drive_Alarm_Active       := #Temp3,
           Freno                    := #Temp4,
           Drive_F_Act              := #RTemp1);
NETWORK
TITLE =
      CALL  "PROFIBUS_MM4" (
           Periferic_Address        := 424,
           Drive_On_Off             := "Comando_M32",
           Drive_Reversing          := FALSE,
           Drive_Fault_ACKN         := FALSE,
           Drive_F_Setpoint         := 5.000000e+01,
           Drive_in_operation       := #Temp1,
           Drive_Fault_Active       := "M67.4",
           Drive_Alarm_Active       := #Temp3,
           Freno                    := #Temp4,
           Drive_F_Act              := #RTemp1);
NETWORK
TITLE =
      CALL  "PROFIBUS_MM4" (
           Periferic_Address        := 436,
           Drive_On_Off             := "Comando_M33",
           Drive_Reversing          := FALSE,
           Drive_Fault_ACKN         := FALSE,
           Drive_F_Setpoint         := 5.000000e+01,
           Drive_in_operation       := #Temp1,
           Drive_Fault_Active       := "M67.5",
           Drive_Alarm_Active       := #Temp3,
           Freno                    := #Temp4,
           Drive_F_Act              := #RTemp1);
NETWORK
TITLE =
      CALL  "PROFIBUS_MM4" (
           Periferic_Address        := 448,
           Drive_On_Off             := "Comando_M34",
           Drive_Reversing          := FALSE,
           Drive_Fault_ACKN         := FALSE,
           Drive_F_Setpoint         := 5.000000e+01,
           Drive_in_operation       := #Temp1,
           Drive_Fault_Active       := "M67.6",
           Drive_Alarm_Active       := #Temp3,
           Freno                    := #Temp4,
           Drive_F_Act              := #RTemp1);
NETWORK
TITLE =
      CALL  "PROFIBUS_MM4" (
           Periferic_Address        := 460,
           Drive_On_Off             := "Comando_M35",
           Drive_Reversing          := FALSE,
           Drive_Fault_ACKN         := FALSE,
           Drive_F_Setpoint         := 5.000000e+01,
           Drive_in_operation       := #Temp1,
           Drive_Fault_Active       := "M67.7",
           Drive_Alarm_Active       := #Temp3,
           Freno                    := #Temp4,
           Drive_F_Act              := #RTemp1);
END_FUNCTION

FUNCTION "Gestione finecorsa" : VOID	// FC 18
VERSION : 0.1
BEGIN
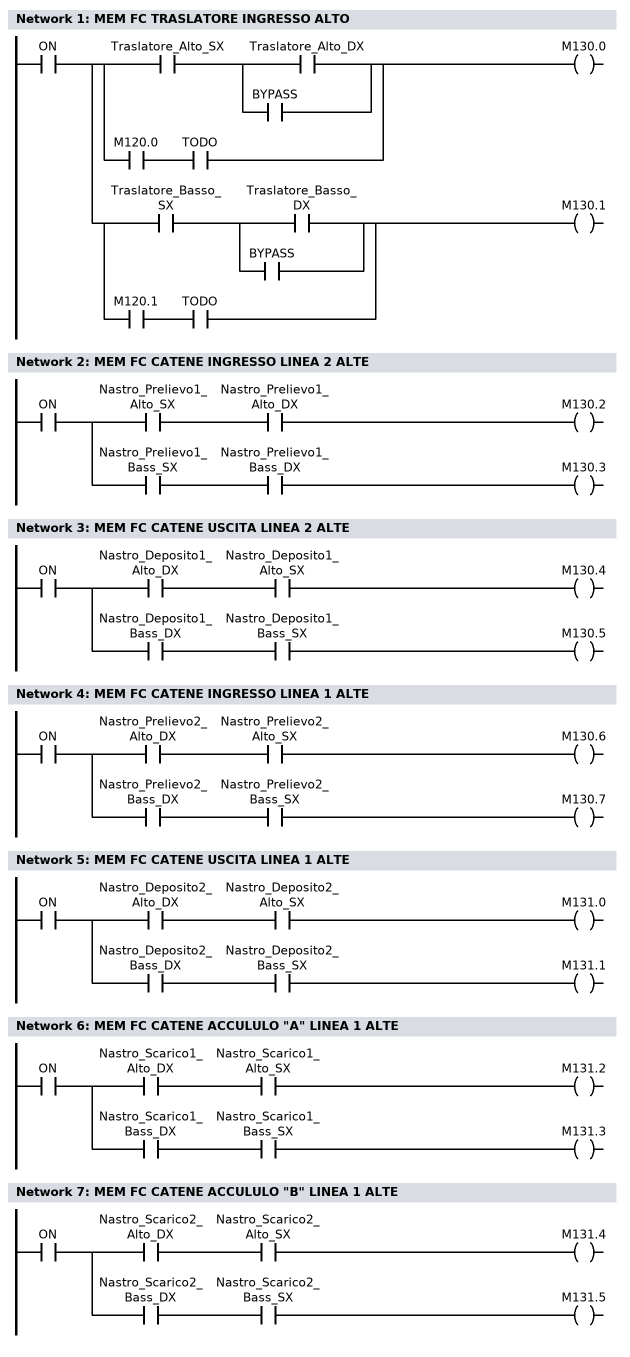
NETWORK
TITLE = MEM FC TRASLATORE INGRESSO ALTO
      A     "ON";
      =     L 0.0;
      A     L 0.0;
      A(;
      A     "Traslatore_Alto_SX";
      A(;
      O     "Traslatore_Alto_DX";
      O     "BYPASS";
      );
      O;
      A     "M120.0";
      A     "TODO";
      );
      =     "M130.0";
      A     L 0.0;
      A(;
      A     "Traslatore_Basso_SX";
      A(;
      O     "Traslatore_Basso_DX";
      O     "BYPASS";
      );
      O;
      A     "M120.1";
      A     "TODO";
      );
      =     "M130.1";
NETWORK
TITLE = MEM FC CATENE INGRESSO LINEA 2 ALTE
      A     "ON";
      =     L 0.0;
      A     L 0.0;
      A     "Nastro_Prelievo1_Alto_SX";
      A     "Nastro_Prelievo1_Alto_DX";
      =     "M130.2";
      A     L 0.0;
      A     "Nastro_Prelievo1_Bass_SX";
      A     "Nastro_Prelievo1_Bass_DX";
      =     "M130.3";
NETWORK
TITLE = MEM FC CATENE USCITA LINEA 2 ALTE
      A     "ON";
      =     L 0.0;
      A     L 0.0;
      A     "Nastro_Deposito1_Alto_DX";
      A     "Nastro_Deposito1_Alto_SX";
      =     "M130.4";
      A     L 0.0;
      A     "Nastro_Deposito1_Bass_DX";
      A     "Nastro_Deposito1_Bass_SX";
      =     "M130.5";
NETWORK
TITLE = MEM FC CATENE INGRESSO LINEA 1 ALTE
      A     "ON";
      =     L 0.0;
      A     L 0.0;
      A     "Nastro_Prelievo2_Alto_DX";
      A     "Nastro_Prelievo2_Alto_SX";
      =     "M130.6";
      A     L 0.0;
      A     "Nastro_Prelievo2_Bass_DX";
      A     "Nastro_Prelievo2_Bass_SX";
      =     "M130.7";
NETWORK
TITLE = MEM FC CATENE USCITA LINEA 1 ALTE
      A     "ON";
      =     L 0.0;
      A     L 0.0;
      A     "Nastro_Deposito2_Alto_DX";
      A     "Nastro_Deposito2_Alto_SX";
      =     "M131.0";
      A     L 0.0;
      A     "Nastro_Deposito2_Bass_DX";
      A     "Nastro_Deposito2_Bass_SX";
      =     "M131.1";
NETWORK
TITLE = MEM FC CATENE ACCULULO "A" LINEA 1 ALTE
      A     "ON";
      =     L 0.0;
      A     L 0.0;
      A     "Nastro_Scarico1_Alto_DX";
      A     "Nastro_Scarico1_Alto_SX";
      =     "M131.2";
      A     L 0.0;
      A     "Nastro_Scarico1_Bass_DX";
      A     "Nastro_Scarico1_Bass_SX";
      =     "M131.3";
NETWORK
TITLE = MEM FC CATENE ACCULULO "B" LINEA 1 ALTE
      A     "ON";
      =     L 0.0;
      A     L 0.0;
      A     "Nastro_Scarico2_Alto_DX";
      A     "Nastro_Scarico2_Alto_SX";
      =     "M131.4";
      A     L 0.0;
      A     "Nastro_Scarico2_Bass_DX";
      A     "Nastro_Scarico2_Bass_SX";
      =     "M131.5";
END_FUNCTION

FUNCTION "Gestione OP" : VOID	// FC 20
VERSION : 0.1
BEGIN
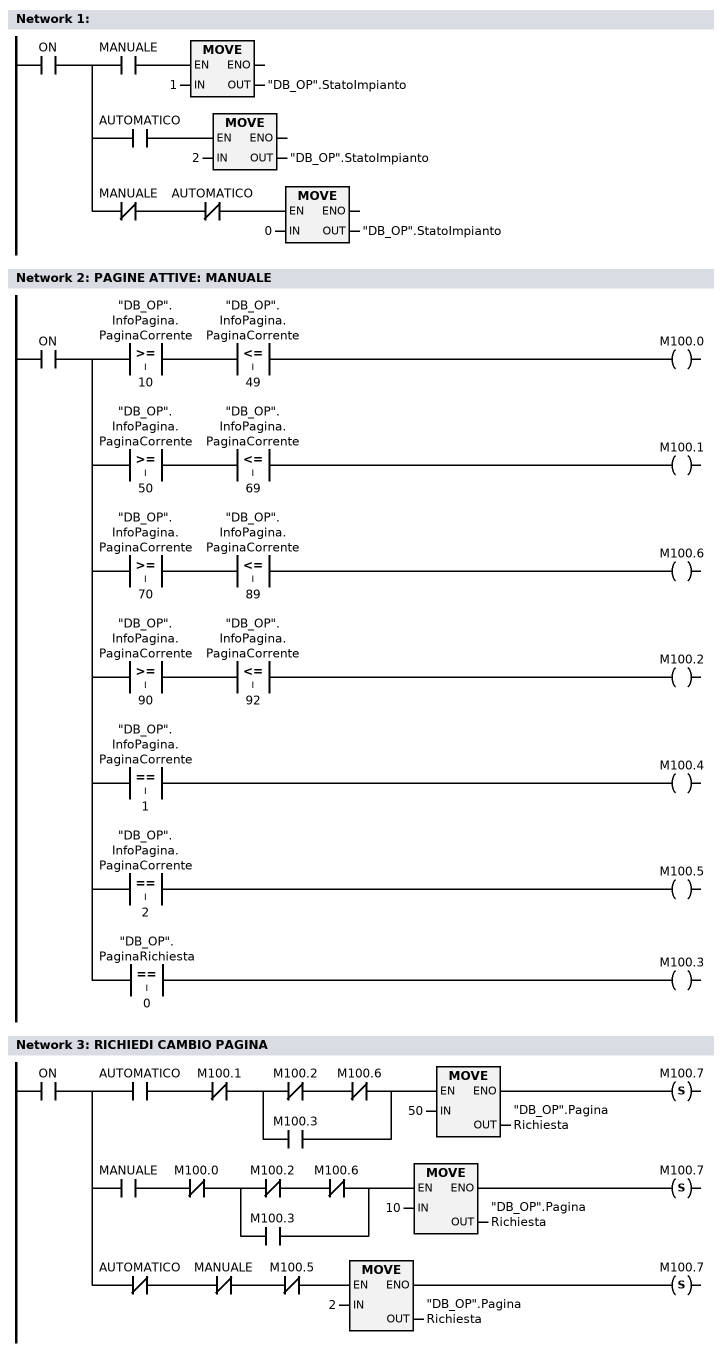
NETWORK
TITLE =
      A     "ON";
      =     L 0.0;
      A     L 0.0;
      A     "MANUALE";
      JNB   _001;
      L     1;
      T     "DB_OP".StatoImpianto;
_001: NOP   0;
      A     L 0.0;
      A     "AUTOMATICO";
      JNB   _002;
      L     2;
      T     "DB_OP".StatoImpianto;
_002: NOP   0;
      A     L 0.0;
      AN    "MANUALE";
      AN    "AUTOMATICO";
      JNB   _003;
      L     0;
      T     "DB_OP".StatoImpianto;
_003: NOP   0;
NETWORK
TITLE = PAGINE ATTIVE: MANUALE
      A     "ON";
      =     L 0.0;
      A     L 0.0;
      A(;
      L     "DB_OP".InfoPagina.PaginaCorrente;
      L     10;
      >=I;
      );
      A(;
      L     "DB_OP".InfoPagina.PaginaCorrente;
      L     49;
      <=I;
      );
      =     "M100.0";
      A     L 0.0;
      A(;
      L     "DB_OP".InfoPagina.PaginaCorrente;
      L     50;
      >=I;
      );
      A(;
      L     "DB_OP".InfoPagina.PaginaCorrente;
      L     69;
      <=I;
      );
      =     "M100.1";
      A     L 0.0;
      A(;
      L     "DB_OP".InfoPagina.PaginaCorrente;
      L     70;
      >=I;
      );
      A(;
      L     "DB_OP".InfoPagina.PaginaCorrente;
      L     89;
      <=I;
      );
      =     "M100.6";
      A     L 0.0;
      A(;
      L     "DB_OP".InfoPagina.PaginaCorrente;
      L     90;
      >=I;
      );
      A(;
      L     "DB_OP".InfoPagina.PaginaCorrente;
      L     92;
      <=I;
      );
      =     "M100.2";
      A     L 0.0;
      A(;
      L     "DB_OP".InfoPagina.PaginaCorrente;
      L     1;
      ==I;
      );
      =     "M100.4";
      A     L 0.0;
      A(;
      L     "DB_OP".InfoPagina.PaginaCorrente;
      L     2;
      ==I;
      );
      =     "M100.5";
      A     L 0.0;
      A(;
      L     "DB_OP".PaginaRichiesta;
      L     0;
      ==I;
      );
      =     "M100.3";
NETWORK
TITLE = RICHIEDI CAMBIO PAGINA
      A     "ON";
      =     L 0.0;
      A     L 0.0;
      A     "AUTOMATICO";
      AN    "M100.1";
      A(;
      AN    "M100.2";
      AN    "M100.6";
      O     "M100.3";
      );
      JNB   _004;
      L     50;
      T     "DB_OP".PaginaRichiesta;
      SET;
      SAVE;
      CLR;
_004: A     BR;
      S     "M100.7";
      A     L 0.0;
      A     "MANUALE";
      AN    "M100.0";
      A(;
      AN    "M100.2";
      AN    "M100.6";
      O     "M100.3";
      );
      JNB   _005;
      L     10;
      T     "DB_OP".PaginaRichiesta;
      SET;
      SAVE;
      CLR;
_005: A     BR;
      S     "M100.7";
      A     L 0.0;
      AN    "AUTOMATICO";
      AN    "MANUALE";
      AN    "M100.5";
      JNB   _006;
      L     2;
      T     "DB_OP".PaginaRichiesta;
      SET;
      SAVE;
      CLR;
_006: A     BR;
      S     "M100.7";
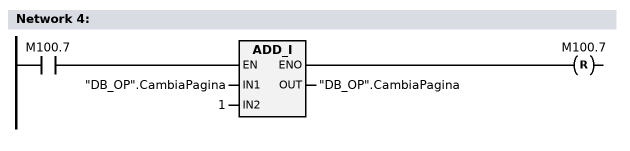
NETWORK
TITLE =
      A     "M100.7";
      JNB   _007;
      L     "DB_OP".CambiaPagina;
      L     1;
      +I;
      T     "DB_OP".CambiaPagina;
      AN    OV;
      SAVE;
      CLR;
_007: A     BR;
      R     "M100.7";
END_FUNCTION

FUNCTION "Gestione Timer e Counter" : VOID	// FC 30
VERSION : 0.1
BEGIN
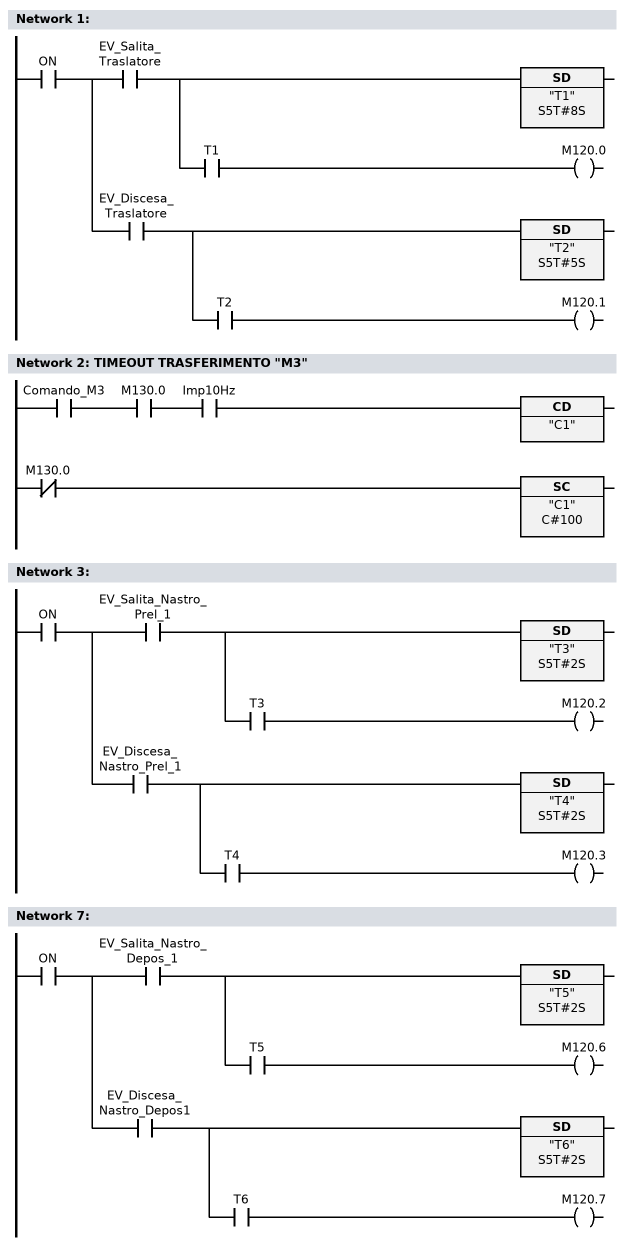
NETWORK
TITLE =
      A     "ON";
      =     L 0.0;
      A     L 0.0;
      A     "EV_Salita_Traslatore";
      =     L 0.1;
      A     L 0.1;
      BLD   102;
      L     S5T#8S;
      SD    "T1";
      A     L 0.1;
      A     "T1";
      =     "M120.0";
      A     L 0.0;
      A     "EV_Discesa_Traslatore";
      =     L 0.1;
      A     L 0.1;
      BLD   102;
      L     S5T#5S;
      SD    "T2";
      A     L 0.1;
      A     "T2";
      =     "M120.1";
NETWORK
TITLE = TIMEOUT TRASFERIMENTO "M3"
      A     "Comando_M3";
      A     "M130.0";
      A     "Imp10Hz";
      CD    "C1";
      BLD   101;
      AN    "M130.0";
      L     C#100;
      S     "C1";
      NOP   0;
      NOP   0;
      NOP   0;
      NOP   0;
NETWORK
TITLE =
      A     "ON";
      =     L 0.0;
      A     L 0.0;
      A     "EV_Salita_Nastro_Prel_1";
      =     L 0.1;
      A     L 0.1;
      BLD   102;
      L     S5T#2S;
      SD    "T3";
      A     L 0.1;
      A     "T3";
      =     "M120.2";
      A     L 0.0;
      A     "EV_Discesa_Nastro_Prel_1";
      =     L 0.1;
      A     L 0.1;
      BLD   102;
      L     S5T#2S;
      SD    "T4";
      A     L 0.1;
      A     "T4";
      =     "M120.3";
NETWORK
TITLE = TEMPO SVUOTAMENTO CATENA INGRESSO CADENZATORE LINEA 2
      A(;
      A     "M21.0";
      A     "Comando_M4";
      A     "Imp10Hz";
      CD    "C2";
      BLD   101;
      AN    "M21.0";
      A     "M120.4";
      L     C#60;
      S     "C2";
      NOP   0;
      NOP   0;
      NOP   0;
      A     "C2";
      );
      NOT;
      =     "M120.4";
NETWORK
TITLE = TEMPO SVUOTAMENTO CATENA INGRESSO CADENZATORE LINEA 2
      A(;
      A     "M20.4";
      A     "Comando_M4";
      A     "M130.2";
      A     "Imp10Hz";
      CD    "C20";
      BLD   101;
      AN    "M20.4";
      L     C#30;
      S     "C20";
      NOP   0;
      NOP   0;
      NOP   0;
      A     "C20";
      );
      NOT;
      =     "M122.5";
NETWORK
TITLE = TEMPO PASSO CATENE LINEA 2
      A(;
      A     "M21.3";
      A     "Comando_M5";
      A     "Imp10Hz";
      CD    "C3";
      BLD   101;
      AN    "M21.3";
      A     "M120.5";
      L     C#8;
      S     "C3";
      NOP   0;
      NOP   0;
      NOP   0;
      A     "C3";
      );
      NOT;
      =     "M120.5";
NETWORK
TITLE =
      A     "ON";
      =     L 0.0;
      A     L 0.0;
      A     "EV_Salita_Nastro_Depos_1";
      =     L 0.1;
      A     L 0.1;
      BLD   102;
      L     S5T#2S;
      SD    "T5";
      A     L 0.1;
      A     "T5";
      =     "M120.6";
      A     L 0.0;
      A     "EV_Discesa_Nastro_Depos1";
      =     L 0.1;
      A     L 0.1;
      BLD   102;
      L     S5T#2S;
      SD    "T6";
      A     L 0.1;
      A     "T6";
      =     "M120.7";
NETWORK
TITLE = TEMPO PASSO CATENE LINEA 2
      A(;
      A     "M24.6";
      A     "Comando_M17";
      A     "Imp10Hz";
      CD    "C4";
      BLD   101;
      AN    "M24.6";
      A     "M121.0";
      L     C#10;
      S     "C4";
      NOP   0;
      NOP   0;
      NOP   0;
      A     "C4";
      );
      NOT;
      =     "M121.0";
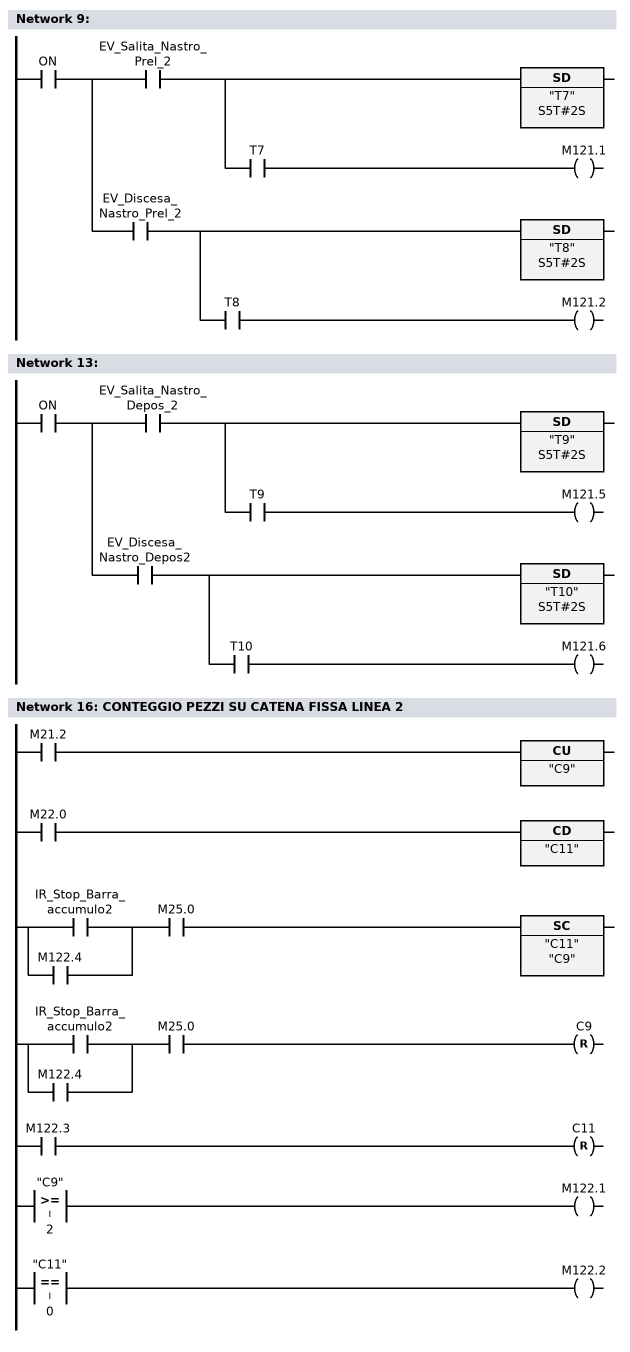
NETWORK
TITLE =
      A     "ON";
      =     L 0.0;
      A     L 0.0;
      A     "EV_Salita_Nastro_Prel_2";
      =     L 0.1;
      A     L 0.1;
      BLD   102;
      L     S5T#2S;
      SD    "T7";
      A     L 0.1;
      A     "T7";
      =     "M121.1";
      A     L 0.0;
      A     "EV_Discesa_Nastro_Prel_2";
      =     L 0.1;
      A     L 0.1;
      BLD   102;
      L     S5T#2S;
      SD    "T8";
      A     L 0.1;
      A     "T8";
      =     "M121.2";
NETWORK
TITLE = TEMPO SVUOTAMENTO CATENA INGRESSO CADENZATORE LINEA 1
      A(;
      A     "M41.0";
      A     "Comando_M11";
      A     "Imp10Hz";
      CD    "C5";
      BLD   101;
      AN    "M41.0";
      A     "M121.3";
      L     C#60;
      S     "C5";
      NOP   0;
      NOP   0;
      NOP   0;
      A     "C5";
      );
      NOT;
      =     "M121.3";
NETWORK
TITLE = RITARDO FUORI INGOMBRO M24
      A(;
      A     "M40.4";
      A     "Comando_M11";
      A     "M130.6";
      A     "Imp10Hz";
      CD    "C21";
      BLD   101;
      AN    "M40.4";
      L     C#30;
      S     "C21";
      NOP   0;
      NOP   0;
      NOP   0;
      A     "C21";
      );
      NOT;
      =     "M122.6";
NETWORK
TITLE = TEMPO PASSO CATENE LINEA 1
      A(;
      A     "M41.3";
      A     "Comando_M10";
      A     "Imp10Hz";
      CD    "C6";
      BLD   101;
      AN    "M41.3";
      A     "M121.4";
      L     C#8;
      S     "C6";
      NOP   0;
      NOP   0;
      NOP   0;
      A     "C6";
      );
      NOT;
      =     "M121.4";
NETWORK
TITLE =
      A     "ON";
      =     L 0.0;
      A     L 0.0;
      A     "EV_Salita_Nastro_Depos_2";
      =     L 0.1;
      A     L 0.1;
      BLD   102;
      L     S5T#2S;
      SD    "T9";
      A     L 0.1;
      A     "T9";
      =     "M121.5";
      A     L 0.0;
      A     "EV_Discesa_Nastro_Depos2";
      =     L 0.1;
      A     L 0.1;
      BLD   102;
      L     S5T#2S;
      SD    "T10";
      A     L 0.1;
      A     "T10";
      =     "M121.6";
NETWORK
TITLE =
      A(;
      A     "M21.1";
      AN    "Proximity_0_Cadenzatore1";
      A     "Comando_M7";
      A     "Imp10Hz";
      CD    "C7";
      BLD   101;
      A     "Proximity_0_Cadenzatore1";
      A     "M121.7";
      L     C#25;
      S     "C7";
      NOP   0;
      NOP   0;
      NOP   0;
      A     "C7";
      );
      NOT;
      =     "M121.7";
NETWORK
TITLE =
      A(;
      A     "M41.1";
      AN    "Proximity_0_Cadenzatore2";
      A     "Comando_M8";
      A     "Imp10Hz";
      CD    "C8";
      BLD   101;
      A     "Proximity_0_Cadenzatore2";
      A     "M122.0";
      L     C#25;
      S     "C8";
      NOP   0;
      NOP   0;
      NOP   0;
      A     "C8";
      );
      NOT;
      =     "M122.0";
NETWORK
TITLE = CONTEGGIO PEZZI SU CATENA FISSA LINEA 2
      A     "M21.2";
      CU    "C9";
      A     "M22.0";
      CD    "C11";
      A(;
      A     "IR_Stop_Barra_accumulo2";
      O     "M122.4";
      );
      A     "M25.0";
      L     "C9";
      S     "C11";
      A(;
      A     "IR_Stop_Barra_accumulo2";
      O     "M122.4";
      );
      A     "M25.0";
      R     "C9";
      A     "M122.3";
      R     "C11";
      L     "C9";
      L     2;
      >=I;
      =     "M122.1";
      L     "C11";
      L     0;
      ==I;
      =     "M122.2";
NETWORK
TITLE =
      A(;
      AN    "M25.0";
      A     "Comando_M6";
      A     "Imp10Hz";
      CD    "C10";
      BLD   101;
      A     "M25.0";
      L     C#60;
      S     "C10";
      NOP   0;
      NOP   0;
      NOP   0;
      A     "C10";
      );
      NOT;
      =     "M122.3";
NETWORK
TITLE =
      A(;
      A     "M25.0";
      A     "Comando_M6";
      A     "Imp10Hz";
      CD    "C12";
      BLD   101;
      AN    "M25.0";
      L     C#80;
      S     "C12";
      NOP   0;
      NOP   0;
      NOP   0;
      A     "C12";
      );
      NOT;
      =     "M122.4";
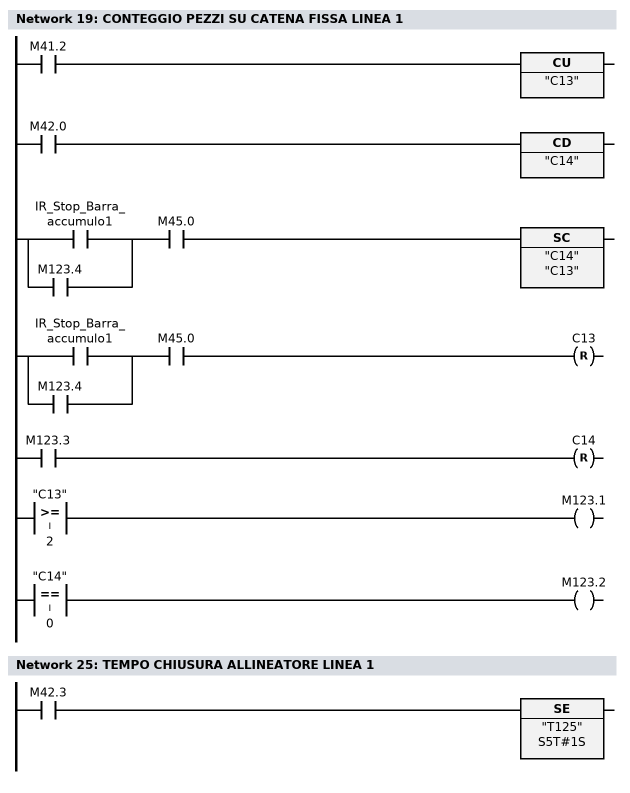
NETWORK
TITLE = CONTEGGIO PEZZI SU CATENA FISSA LINEA 1
      A     "M41.2";
      CU    "C13";
      A     "M42.0";
      CD    "C14";
      A(;
      A     "IR_Stop_Barra_accumulo1";
      O     "M123.4";
      );
      A     "M45.0";
      L     "C13";
      S     "C14";
      A(;
      A     "IR_Stop_Barra_accumulo1";
      O     "M123.4";
      );
      A     "M45.0";
      R     "C13";
      A     "M123.3";
      R     "C14";
      L     "C13";
      L     2;
      >=I;
      =     "M123.1";
      L     "C14";
      L     0;
      ==I;
      =     "M123.2";
NETWORK
TITLE =
      A(;
      AN    "M45.0";
      A     "Comando_M9";
      A     "Imp10Hz";
      CD    "C15";
      BLD   101;
      A     "M45.0";
      L     C#45;
      S     "C15";
      NOP   0;
      NOP   0;
      NOP   0;
      A     "C15";
      );
      NOT;
      =     "M123.3";
NETWORK
TITLE =
      A(;
      A     "M45.0";
      A     "Comando_M9";
      A     "Imp10Hz";
      CD    "C16";
      BLD   101;
      AN    "M45.0";
      L     C#140;
      S     "C16";
      NOP   0;
      NOP   0;
      NOP   0;
      A     "C16";
      );
      NOT;
      =     "M123.4";
NETWORK
TITLE =
      A(;
      A     "M44.1";
      A     "Comando_M12";
      A     "Imp10Hz";
      CD    "C17";
      BLD   101;
      AN    "M44.1";
      L     C#10;
      S     "C17";
      NOP   0;
      NOP   0;
      NOP   0;
      A     "C17";
      );
      NOT;
      =     "M123.5";
NETWORK
TITLE = TEMPO PASSO CATENE LINEA 2
      A(;
      A     "M26.4";
      A     "Comando_M19";
      A     "Imp10Hz";
      CD    "C18";
      BLD   101;
      AN    "M26.4";
      A     "M123.6";
      L     C#10;
      S     "C18";
      NOP   0;
      NOP   0;
      NOP   0;
      A     "C18";
      );
      NOT;
      =     "M123.6";
NETWORK
TITLE =
      A(;
      A     "M45.4";
      A     "Comando_M14";
      A     "Imp10Hz";
      CD    "C19";
      BLD   101;
      AN    "M45.4";
      L     C#10;
      S     "C19";
      NOP   0;
      NOP   0;
      NOP   0;
      A     "C19";
      );
      NOT;
      =     "M123.7";
NETWORK
TITLE = TEMPO CHIUSURA ALLINEATORE LINEA 1
      A     "M42.3";
      L     S5T#1S;
      SE    "T125";
END_FUNCTION

FUNCTION "AG_SEND" : VOID	// FC 106
AUTHOR : SIMATIC
FAMILY : CP_300
NAME : AG_SEND
VERSION : 4.2
VAR_INPUT
  ACT : BOOL ;	// Activate job
  ID { S7_co := 'agag'; S7_server1 := 'connection' }: INT ;	// Connection ID 1..16
  LADDR { S7_co := 'agag'; S7_server1 := 'connection' }: WORD ;	// Module address in hardware configuration
  SEND : ANY ;	// Data destination
  LEN : INT ;	// Buffer for send data
END_VAR
VAR_OUTPUT
  DONE : BOOL ;	// Job done without errors
  ERROR : BOOL ;	// ERROR code
  STATUS : WORD ;	// STATUS code
END_VAR
VAR_TEMP
  LBUSY : BOOL ;	// SFC READ/WRITE Fertigmeldung
  STATIC : BOOL ;
  GEN_DS_LESEN : BOOL ;
  SEND_BUSY : BOOL ;
  SEND_CONF : BOOL ;
  SEND_IN_PROGRESS : BOOL ;
  OFFSETTING : BOOL ;
  READING : BOOL ;
  TEMP_DATA : DWORD ;
  OFFSET : WORD ;
  DIFF : WORD ;
  DS_NR : BYTE ;	// Datensatznummer, SFC Input Parameter
  CON_INF : BYTE ;	// Speicher fuer Quittung vom CP
  RET_WT_STORE : INT ;	// Dynamische Speicher fuer RET_VAL
// (Output Par. des SFCs)
  STORE : ANY ;
  AR1_STORE : DWORD ;
  AR2_STORE : DWORD ;
  FC_DATA_LEN : WORD ;	// Vom Anwender projektrierte Transfer Laenge
  LOOP_COUNT : WORD ;
END_VAR
BEGIN
NETWORK
TITLE =
      TAR1  #AR1_STORE;
      TAR2  #AR2_STORE;
      L     0;
      T     #STATUS;
      SET;
      R     #ERROR;
      R     #DONE;
      R     #STATIC;
      R     #GEN_DS_LESEN;
      R     #SEND_BUSY;
      R     #SEND_CONF;
      R     #SEND_IN_PROGRESS;
      R     #OFFSETTING;
      R     #READING;
      L     1;
      L     #ID;
      >I;
      JC    NKO;
      L     16;
      <=I;
      JC    NOK;
NKO:  L     W#16#8186;
      JU    ERRS;
NOK:  L     #LADDR;
      SLD   3;
      LAR1;
      L     PIW [AR1,P#4.0];
      SRW   7;
      JZ    STAA;
      SRW   1;
      JZ    GEN1;
STAA: SET;
      S     #STATIC;
      L     #ID;
      DEC   1;
      SRW   2;
      SLW   1;
      L     #LADDR;
      +I;
      INC   8;
      SLD   3;
      LAR1;
      L     #ID;
      DEC   1;
      SRW   2;
      L     PIW [AR1,P#0.0];
      JZ    UG;
      JU    M5;
UG:   SRW   8;
M5:   L     #ID;
      SRW   1;
      JP    UGR;
      TAK;
      SRW   6;
      JU    GER;
UGR:  TAK;
      SRW   2;
GER:  L     B#16#3;
      AW;
      L     1;
      ==I;
      JC    BUSY;
      TAK;
      L     2;
      ==I;
      JC    ABG;
      TAK;
      L     0;
      ==I;
      JC    CONT;
      A     #ACT;
      L     W#16#8183;
      JC    ERRS;
      SET;
      SAVE;
      L     0;
      JU    END;
GEN1: L     #ID;
      DEC   1;
      L     1;
      SLW;
      L     PID [AR1,P#10.0];
      T     #TEMP_DATA;
      AW;
      JP    SBSY;
      JU    NXT;
SBSY: S     #SEND_BUSY;
NXT:  TAK;
      L     #TEMP_DATA;
      SRD   16;
      AW;
      JP    SCNF;
      JU    NXTT;
SCNF: S     #SEND_CONF;
NXTT: A     #SEND_BUSY;
      A     #SEND_CONF;
      S     #SEND_IN_PROGRESS;
      JC    CNT;
      A     #SEND_BUSY;
      JC    BUSY;
      A     #SEND_CONF;
      JC    ABG;
CONT: A     #ACT;
      JC    CNT;
      SET;
      SAVE;
      L     0;
      JU    END;
CNT:  L     #ID;
      L     15;
      +I;
      T     #DS_NR;
      L     P##SEND;
      LAR2;
      L     B [AR2,P#1.0];
      L     2;
      <>I;
      TAK;
      JC    WRD;
      L     W [AR2,P#2.0];
      JU    BITE;
WRD:  L     4;
      <>I;
      TAK;
      JC    DWRD;
      L     W [AR2,P#2.0];
      SLW   1;
      JU    BITE;
DWRD: L     6;
      ==I;
      TAK;
      JC    TYDW;
      L     W#16#8184;
      JU    ERRS;
TYDW: L     W [AR2,P#2.0];
      SLW   2;
BITE: T     #FC_DATA_LEN;
      L     #LEN;
      L     #FC_DATA_LEN;
      <=I;
      JC    LVST;
      L     W#16#8185;
      JU    ERRS;
LVST: TAK;
      T     #FC_DATA_LEN;
      SRD   16;
      JZ    LOKK;
      L     W#16#8F22;
      JU    ERRS;
LOKK: AN    #STATIC;
      JC    HSDL;
      L     P##SEND;
      LAR1;
      L     P##STORE;
      LAR2;
      L     W#16#1002;
      T     LW [AR2,P#0.0];
      L     W [AR1,P#4.0];
      T     LW [AR2,P#4.0];
      L     #FC_DATA_LEN;
      T     LW [AR2,P#2.0];
      L     D [AR1,P#6.0];
      T     LD [AR2,P#6.0];
      A     #STATIC;
      JC    TTT;
HSDL: L     #LADDR;
      SLD   3;
      LAR1;
      A     #READING;
      L     B#16#76;
      JC    III;
      L     B#16#7E;
III:  L     #DS_NR;
      SLW   8;
      OW;
      SLD   16;
      L     #FC_DATA_LEN;
      OD;
      T     PQD [AR1,P#4.0];
      L     250;
STRT: T     #LOOP_COUNT;
      L     PID [AR1,P#4.0];
      T     #TEMP_DATA;
      SRD   17;
      JZ    VAL;
      SRW   3;
      JZ    RECX;
      A     #READING;
      JC    WEIT;
      JU    DOKK;
RECX: AN    #READING;
      JC    WEIT;
DOKK: L     #TEMP_DATA;
      SRD   21;
      JZ    DDD;
      JU    WEIT;
DDD:  SRW   3;
      L     #DS_NR;
      <>I;
      JC    WEIT;
      JU    LGBY;
WEIT: L     #LOOP_COUNT;
      LOOP  STRT;
      L     W#16#80C4;
      T     #RET_WT_STORE;
      JU    ERRR;
LGBY: L     #TEMP_DATA;
      SRD   19;
      JZ    NSQ;
      SET;
      S     #OFFSETTING;
      JU    ERRR;
NSQ:  L     #TEMP_DATA;
      T     #RET_WT_STORE;
      JU    ERRR;
VAL:  SET;
      L     #TEMP_DATA;
      SRD   20;
      JZ    RECV;
      A     #READING;
      AN    #SEND_IN_PROGRESS;
      L     W#16#80C2;
      JC    ERRS;
      A     #READING;
      JC    BUSY;
      JU    DOK;
RECV: AN    #READING;
      AN    #SEND_IN_PROGRESS;
      L     W#16#80C2;
      JC    ERRS;
      AN    #READING;
      JC    BUSY;
DOK:  L     #TEMP_DATA;
      SRD   24;
      L     #DS_NR;
      ==I;
      JC    DSOK;
      A     #SEND_IN_PROGRESS;
      JC    BUSY;
      L     W#16#80C2;
      JU    ERRS;
DSOK: A     #READING;
      JC    RET1;
      L     #FC_DATA_LEN;
      L     #TEMP_DATA;
      T     #OFFSET;
      -I;
      T     #DIFF;
      L     240;
      <=I;
      JC    BBC;
      T     #DIFF;
BBC:  L     P##SEND;
      LAR1;
      L     P##STORE;
      LAR2;
      L     W#16#1002;
      T     LW [AR2,P#0.0];
      L     #DIFF;
      T     LW [AR2,P#2.0];
      L     W [AR1,P#4.0];
      T     LW [AR2,P#4.0];
      L     D [AR1,P#6.0];
      L     #OFFSET;
      SLD   3;
      +D;
      T     LD [AR2,P#6.0];
TTT:  CALL  "WR_REC" (
           REQ                      := TRUE,
           IOID                     := B#16#54,
           LADDR                    := #LADDR,
           RECNUM                   := #DS_NR,
           RECORD                   := #STORE,
           RET_VAL                  := #RET_WT_STORE,
           BUSY                     := #LBUSY);
      L     #RET_WT_STORE;
      L     W#16#F00;
      AW;
      TAK;
      JZ    EEA;
      L     W#16#F00;
      OW;
      T     #RET_WT_STORE;
EEA:  A     #STATIC;
      JC    LLL;
      A     #LBUSY;
      =     #OFFSETTING;
      L     #RET_WT_STORE;
      L     0;
      ==I;
      JC    BUSY;
SFCE: L     #LADDR;
      SLD   3;
      LAR1;
      L     PID [AR1,P#4.0];
      SRD   18;
      L     #RET_WT_STORE;
      JZ    ERRS;
ERRR: L     #LADDR;
      SLD   3;
      LAR1;
      AN    #OFFSETTING;
      JC    GGG;
      A     #READING;
      L     B#16#74;
      JC    HHH;
      L     B#16#7C;
      JU    HHH;
GGG:  A     #READING;
      L     B#16#70;
      JC    HHH;
      L     B#16#78;
HHH:  L     #DS_NR;
      SLW   8;
      OW;
      SLD   16;
      L     #FC_DATA_LEN;
      OD;
      T     PQD [AR1,P#4.0];
      L     250;
STR2: T     #LOOP_COUNT;
      L     PID [AR1,P#4.0];
      T     #TEMP_DATA;
      SRD   17;
      JZ    STA;
      SRW   4;
      JZ    STA;
      JU    BREK;
STA:  L     #TEMP_DATA;
      SRD   20;
      JZ    RECC;
      A     #READING;
      JC    BREK;
      JU    DROK;
RECC: AN    #READING;
      JC    BREK;
DROK: SRW   4;
      L     #DS_NR;
      <>I;
      JC    BREK;
      L     #LOOP_COUNT;
      LOOP  STR2;
      L     W#16#80C4;
      JU    ERRS;
BREK: A     #OFFSETTING;
      JC    BUSY;
      L     #RET_WT_STORE;
      JU    ERRS;
LLL:  A     #LBUSY;
      JC    BUSY;
      L     0;
      L     #RET_WT_STORE;
      ==I;
      JC    BUSY;
      JU    ERRS;
      JU    END;
ABG:  S     #READING;
      L     #ID;
      L     31;
      +I;
      T     #DS_NR;
      A     #STATIC;
      JC    RET1;
      L     1;
      T     #FC_DATA_LEN;
      JU    HSDL;
RET1: CALL  "RD_REC" (
           REQ                      := TRUE,
           IOID                     := B#16#54,
           LADDR                    := #LADDR,
           RECNUM                   := #DS_NR,
           RET_VAL                  := #RET_WT_STORE,
           BUSY                     := #LBUSY,
           RECORD                   := #CON_INF);
      A     #STATIC;
      JC    KKK;
      A     #LBUSY;
      =     #OFFSETTING;
      L     #RET_WT_STORE;
      L     0;
      <>I;
      JC    SFCE;
      JU    REOK;
KKK:  A     #LBUSY;
      JC    BUSY;
      L     0;
      L     #RET_WT_STORE;
      ==I;
      JC    REOK;
      L     W#16#F00;
      AW;
      TAK;
      JZ    ERRS;
      L     W#16#F00;
      OW;
      JU    ERRS;
REOK: L     0;
      L     #CON_INF;
      ==I;
      JC    NUL;
      L     B#16#83;
      ==I;
      L     W#16#8183;
      JC    ERRS;
      L     #CON_INF;
      L     W#16#8300;
      OW;
      JU    ERRS;
NUL:  SET;
      A     #STATIC;
      JC    AOK;
      L     #LADDR;
      SLD   3;
      LAR1;
      L     250;
NX:   T     #LOOP_COUNT;
      L     #ID;
      DEC   1;
      L     1;
      SLW;
      L     PID [AR1,P#10.0];
      SRD   16;
      AW;
      JZ    AOK;
      L     #LOOP_COUNT;
      LOOP  NX;
      L     W#16#80C4;
      JU    ERRS;
AOK:  SET;
      S     #DONE;
      SAVE;
      L     0;
      JU    END;
ERRS: SET;
      S     #ERROR;
      CLR;
      SAVE;
      JU    END;
BUSY: SET;
      SAVE;
      L     W#16#8181;
END:  T     #STATUS;
      LAR1  #AR1_STORE;
      LAR2  #AR2_STORE;
      BEU;
NETWORK
TITLE =
END_FUNCTION

FUNCTION "AG_RECV" : VOID	// FC 107
AUTHOR : SIMATIC
FAMILY : CP_300
NAME : AG_RECV
VERSION : 4.7
VAR_INPUT
  ID { S7_co := 'agag'; S7_server1 := 'connection' }: INT ;	// Connection ID 1..16
  LADDR { S7_co := 'agag'; S7_server1 := 'connection' }: WORD ;	// Module address in hardware configuration
  RECV : ANY ;	// Buffer for received data
END_VAR
VAR_OUTPUT
  NDR : BOOL ;	// Indicates whether new data were received
  ERROR : BOOL ;	// ERROR code
  STATUS : WORD ;	// STATUS code
  LEN : INT ;	// Number of received bytes
END_VAR
VAR_TEMP
  LBUSY : BOOL ;	// SFC READ/WRITE Fertigmeldung
  STATIC : BOOL ;
  OFFSETTING : BOOL ;
  DS_NR : BYTE ;	// Datensatznummer, SFC Input Parameter
  RET_WT_STORE : INT ;	// Dynamische Speicher fuer RET_VAL
// (Output Par. des SFCs)
  STORE : ANY ;
  AR1_STORE : DWORD ;
  AR2_STORE : DWORD ;
  DATA_LEN : WORD ;
  FC_DATA_LEN : WORD ;	// Vom Anwender projektrierte Transfer Laenge
  LOOP_COUNT : WORD ;
  TEMP_DATA : DWORD ;
  OFFSET : WORD ;
  DIFF : WORD ;
END_VAR
BEGIN
NETWORK
TITLE =
      TAR1  #AR1_STORE;
      TAR2  #AR2_STORE;
      L     0;
      T     #STATUS;
      T     #LEN;
      T     #OFFSET;
      SET;
      R     #ERROR;
      R     #STATIC;
      R     #NDR;
      R     #OFFSETTING;
      R     #LBUSY;
      L     1;
      L     #ID;
      >I;
      JC    NKO;
      L     16;
      <=I;
      JC    NOK;
NKO:  L     W#16#8186;
      JU    ERRS;
NOK:  L     #LADDR;
      SLD   3;
      LAR1;
      L     PIW [AR1,P#4.0];
      SRW   7;
      JZ    STAA;
      SRW   1;
      JZ    GEN1;
STAA: SET;
      S     #STATIC;
      L     #ID;
      DEC   1;
      SRW   2;
      SLW   1;
      L     #LADDR;
      +I;
      INC   8;
      SLD   3;
      LAR1;
      L     #ID;
      DEC   1;
      SRW   2;
      L     PIW [AR1,P#0.0];
      JZ    UG;
      JU    M5;
UG:   SRW   8;
M5:   L     #ID;
      SRW   1;
      JP    UGR;
      TAK;
      SRW   4;
      JU    GER;
UGR:  TAK;
GER:  L     B#16#3;
      AW;
      L     0;
      ==I;
      JC    CONT;
      TAK;
      L     1;
      ==I;
      JC    BUSY;
      TAK;
      L     2;
      ==I;
      L     W#16#8184;
      JC    ERRS;
      L     W#16#8183;
      JU    ERRS;
GEN1: L     #ID;
      DEC   1;
      L     1;
      SLW;
      L     PIW [AR1,P#14.0];
      AW;
      JP    BUSY;
CONT: L     #ID;
      L     15;
      +I;
      T     #DS_NR;
      L     P##RECV;
      LAR2;
      L     B [AR2,P#1.0];
      L     2;
      <>I;
      TAK;
      JC    WRD;
      L     W [AR2,P#2.0];
      JU    BITE;
WRD:  L     4;
      <>I;
      TAK;
      JC    DWRD;
      L     W [AR2,P#2.0];
      SLW   1;
      JU    BITE;
DWRD: L     6;
      ==I;
      TAK;
      JC    TYDW;
      L     W#16#8184;
      JU    ERRS;
TYDW: L     W [AR2,P#2.0];
      SLW   2;
BITE: T     #FC_DATA_LEN;
      A     #STATIC;
      JC    BBB;
      L     0;
      <I;
      TAK;
      L     W#16#8F23;
      JC    ERRS;
      TAK;
      L     0;
      ==I;
      L     W#16#8F7F;
      JC    ERRS;
      L     #LADDR;
      SLD   3;
      LAR1;
      L     B#16#76;
      L     #DS_NR;
      SLW   8;
      OW;
      SLD   16;
      L     #FC_DATA_LEN;
      OD;
      T     PQD [AR1,P#4.0];
      L     250;
STRT: T     #LOOP_COUNT;
      L     PID [AR1,P#4.0];
      T     #TEMP_DATA;
      SRD   17;
      JZ    VAL;
      SRW   3;
      JZ    JJJ;
      JU    WEIT;
JJJ:  SRW   1;
      JZ    DDD;
      JU    WEIT;
DDD:  SRW   3;
      L     #DS_NR;
      <>I;
      JC    WEIT;
      JU    LGBY;
WEIT: L     #LOOP_COUNT;
      LOOP  STRT;
      L     W#16#80C4;
      T     #RET_WT_STORE;
      JU    ERRR;
LGBY: L     #TEMP_DATA;
      SRD   19;
      JZ    NSQ;
      SET;
      S     #OFFSETTING;
      JU    ERRR;
NSQ:  L     #TEMP_DATA;
      T     #RET_WT_STORE;
      JU    ERRR;
VAL:  L     #TEMP_DATA;
      SRD   20;
      JZ    OKK;
      JU    BUSY;
OKK:  SRW   4;
      L     #DS_NR;
      <>I;
      JC    BUSY;
      L     PIW [AR1,P#8.0];
      T     #FC_DATA_LEN;
      L     #TEMP_DATA;
      T     #OFFSET;
      -I;
      T     #DIFF;
      L     240;
      <=I;
      JC    BBB;
      T     #DIFF;
BBB:  L     P##RECV;
      LAR1;
      L     P##STORE;
      LAR2;
      L     W [AR1,P#4.0];
      T     LW [AR2,P#4.0];
      A     #STATIC;
      JC    JJU;
      L     W#16#1002;
      T     LW [AR2,P#0.0];
      L     #DIFF;
      T     LW [AR2,P#2.0];
      L     D [AR1,P#6.0];
      L     #OFFSET;
      SLD   3;
      +D;
      T     LD [AR2,P#6.0];
      L     #DIFF;
      L     0;
      ==I;
      JC    ERRR;
      JU    JJR;
JJU:  L     D [AR1,P#0.0];
      T     LD [AR2,P#0.0];
      L     D [AR1,P#6.0];
      T     LD [AR2,P#6.0];
JJR:  CALL  "RD_REC" (
           REQ                      := TRUE,
           IOID                     := B#16#54,
           LADDR                    := #LADDR,
           RECNUM                   := #DS_NR,
           RET_VAL                  := #RET_WT_STORE,
           BUSY                     := #LBUSY,
           RECORD                   := #STORE);
      A     #LBUSY;
      A     #STATIC;
      JC    BUSY;
      L     #RET_WT_STORE;
      L     W#16#F00;
      AW;
      TAK;
      JZ    EEA;
      L     W#16#F00;
      OW;
      T     #RET_WT_STORE;
EEA:  A     #LBUSY;
      =     #OFFSETTING;
      L     #RET_WT_STORE;
      L     0;
      <>I;
      AN    #STATIC;
      JC    SFCE;
      <>I;
      TAK;
      JC    ERRS;
      A     #STATIC;
      JC    REOK;
      L     #OFFSET;
      L     #DIFF;
      +I;
      L     #FC_DATA_LEN;
      >=I;
      TAK;
      T     #LEN;
      JC    LOK;
      JU    BUSY;
SFCE: L     #LADDR;
      SLD   3;
      LAR1;
      L     PID [AR1,P#4.0];
      SRD   18;
      L     #RET_WT_STORE;
      JZ    END;
ERRR: L     #FC_DATA_LEN;
      L     #TEMP_DATA;
      -I;
      T     #DIFF;
      L     240;
      <=I;
      JC    KOSE;
      T     #DIFF;
KOSE: L     #DIFF;
      L     0;
      <>I;
      JC    WEER;
      S     #OFFSETTING;
WEER: L     #LADDR;
      SLD   3;
      LAR1;
      AN    #OFFSETTING;
      JC    GGG;
      L     B#16#74;
      JU    HHH;
GGG:  L     B#16#70;
HHH:  L     #DS_NR;
      SLW   8;
      OW;
      SLD   16;
      L     #FC_DATA_LEN;
      OD;
      T     PQD [AR1,P#4.0];
      L     250;
STR2: T     #LOOP_COUNT;
      L     PID [AR1,P#4.0];
      T     #TEMP_DATA;
      SRD   17;
      JZ    STA;
      SRW   4;
      JZ    STA;
      JU    BREK;
STA:  L     #TEMP_DATA;
      SRD   20;
      JZ    AAA;
      JU    BREK;
AAA:  SRW   4;
      L     #DS_NR;
      <>I;
      JC    BREK;
      L     #LOOP_COUNT;
      LOOP  STR2;
      L     W#16#80C4;
      JU    ERRS;
BREK: L     #DIFF;
      L     0;
      ==I;
      JC    LOK;
      A     #OFFSETTING;
      JC    BUSY;
      L     W#16#8181;
      L     #RET_WT_STORE;
      <>I;
      JC    ERRS;
      TAK;
      JU    END;
REOK: L     #LADDR;
      SLD   3;
      LAR1;
      L     PIW [AR1,P#6.0];
      SRW   8;
      T     #LEN;
      L     #FC_DATA_LEN;
      <=I;
      JC    LOK;
      L     W#16#8185;
      JU    ERRS;
LOK:  SET;
      S     #NDR;
      SAVE;
      L     0;
      JU    END;
ERRS: SET;
      S     #ERROR;
      CLR;
      SAVE;
      JU    END;
BUSY: SET;
      SAVE;
      L     W#16#8180;
END:  T     #STATUS;
      LAR1  #AR1_STORE;
      LAR2  #AR2_STORE;
      BEU;
NETWORK
TITLE =
END_FUNCTION

// FC 200: know-how protected block, not included

FUNCTION "FC_AllarmeAttivo" : BOOL	// FC 201
VERSION : 0.0
VAR_OUTPUT
  RET_VAL : BOOL ;
END_VAR
VAR_IN_OUT
  Allarmi : STRUCT
   Msg_001 : BOOL ;	//INTERVENTO TERMICO "KMC1" (E0.0)
   Msg_002 : BOOL ;	//INTERVENTO TERMICO "KMC2" (E0.1)
   Msg_003 : BOOL ;	//INTERVENTO TERMICO "KMC3" (E0.2)
   Msg_004 : BOOL ;	//INTERVENTO TERMICO "KMC4" (E0.3)
   Msg_005 : BOOL ;	//INTERVENTO TERMICO "KMC5" (E0.4)
   Msg_006 : BOOL ;	//INTERVENTO TERMICO "KMC6" (E0.5)
   Msg_007 : BOOL ;	//INTERVENTO TERMICO "KMC7" (E0.6)
   Msg_008 : BOOL ;	//INTERVENTO TERMICO "KMC8" (E0.7)
   Msg_009 : BOOL ;	//INTERVENTO TERMICO "KMC9" (E1.0)
   Msg_010 : BOOL ;	//INTERVENTO TERMICO "KMC10" (E1.1)
   Msg_011 : BOOL ;	//INTERVENTO TERMICO "KMC11" (E1.2)
   Msg_012 : BOOL ;	//INTERVENTO TERMICO "KMC12" (E1.3)
   Msg_013 : BOOL ;	//INTERVENTO TERMICO "KMC13" (E1.4)
   Msg_014 : BOOL ;	//INTERVENTO TERMICO "KMC14" (E1.5)
   Msg_015 : BOOL ;	//INTERVENTO TERMICO "KMC15" (E1.6)
   Msg_016 : BOOL ;	//INTERVENTO TERMICO "KMC16" (E1.7)
   Msg_017 : BOOL ;	//INTERVENTO TERMICO "KMC17" (E2.0)
   Msg_018 : BOOL ;	//INTERVENTO TERMICO "KMC18" (E2.1)
   Msg_019 : BOOL ;	//INTERVENTO TERMICO "KMC19" (E2.2)
   Msg_020 : BOOL ;	//INTERVENTO TERMICO "KMC20" (E2.3)
   Msg_021 : BOOL ;	//INTERVENTO TERMICO "QF20" ALIM. INVERTER A1 "M20" (E3.0)
   Msg_022 : BOOL ;	//INTERVENTO TERMICO "QF21" ALIM. INVERTER A2 "M21" (E3.1)
   Msg_023 : BOOL ;	//INTERVENTO TERMICO "QF22" ALIM. INVERTER A3 "M22" (E3.2)
   Msg_024 : BOOL ;	//INTERVENTO TERMICO "QF23" ALIM. INVERTER A4 "M23" (E3.3)
   Msg_025 : BOOL ;	//INTERVENTO TERMICO "QF24" ALIM. INVERTER A5 "M24" (E3.4)
   Msg_026 : BOOL ;	//INTERVENTO TERMICO "QF25" ALIM. INVERTER A6 "M25" (E3.5)
   Msg_027 : BOOL ;	//INTERVENTO TERMICO "QF26" ALIM. INVERTER A7 "M26" (E3.6)
   Msg_028 : BOOL ;	//INTERVENTO TERMICO "QF27" ALIM. INVERTER A8 "M27" (E3.7)
   Msg_029 : BOOL ;	//INTERVENTO TERMICO "QF28" ALIM. INVERTER A9 "M28" (E4.0)
   Msg_030 : BOOL ;	//INTERVENTO TERMICO "QF29" ALIM. INVERTER A10 "M29" (E4.1)
   Msg_031 : BOOL ;	//INTERVENTO TERMICO "QF30" ALIM. INVERTER A11 "M30" (E4.2)
   Msg_032 : BOOL ;	//INTERVENTO TERMICO "QF31" ALIM. INVERTER A12 "M31" (E4.3)
   Msg_033 : BOOL ;	//INTERVENTO TERMICO "QF32" ALIM. INVERTER A13 "M32" (E4.4)
   Msg_034 : BOOL ;	//INTERVENTO TERMICO "QF33" ALIM. INVERTER A14 "M33" (E4.5)
   Msg_035 : BOOL ;	//INTERVENTO TERMICO "QF34" ALIM. INVERTER A15 "M34" (E4.6)
   Msg_036 : BOOL ;	//INTERVENTO TERMICO "QF35" ALIM. INVERTER A16 "M35" (E4.7)
   Msg_037 : BOOL ;	//INTERVENTO TERMICO "QF36"(E5.0)
   Msg_038 : BOOL ;
   Msg_039 : BOOL ;
   Msg_040 : BOOL ;
   Msg_041 : BOOL ;	//INTERVENTO PROTEZIONE "QF6" VENTILAZIONE QUADRO (E5.1)
   Msg_042 : BOOL ;	//INTERVENTO PROTEZIONE "QF8"  (E5.2)
   Msg_043 : BOOL ;	//INTERVENTO PROTEZIONE "QF19" ALIM. CIRCUITI D'EMERGENZA  (E5.3)
   Msg_044 : BOOL ;	//INTERVENTO PROTEZIONE "QF10" ALIM. COMANDI QUADRO (E5.4)
   Msg_045 : BOOL ;	//INTERVENTO PROTEZIONE "QF11" ALIM. COMANDI JP1  (E5.5)
   Msg_046 : BOOL ;	//INTERVENTO PROTEZIONE "QF12" ALIM. COMANDI JP2  (E5.6)
   Msg_047 : BOOL ;	//INTERVENTO PROTEZIONE "QF13" ALIM. COMANDI JP3  (E5.7)
   Msg_048 : BOOL ;
   Msg_049 : BOOL ;	//FAULT NODO PROFIBUS 3 (INVERTER "M20")
   Msg_050 : BOOL ;	//FAULT NODO PROFIBUS 4 (INVERTER "M21")
   Msg_051 : BOOL ;	//FAULT NODO PROFIBUS 5 (INVERTER "M22")
   Msg_052 : BOOL ;	//FAULT NODO PROFIBUS 6 (INVERTER "M23")
   Msg_053 : BOOL ;	//FAULT NODO PROFIBUS 7 (INVERTER "M24")
   Msg_054 : BOOL ;	//FAULT NODO PROFIBUS 8 (INVERTER "M25")
   Msg_055 : BOOL ;	//FAULT NODO PROFIBUS 9 (INVERTER "M26")
   Msg_056 : BOOL ;	//FAULT NODO PROFIBUS 10 (INVERTER "M27")
   Msg_057 : BOOL ;	//FAULT NODO PROFIBUS 11 (INVERTER "M28")
   Msg_058 : BOOL ;	//FAULT NODO PROFIBUS 12 (INVERTER "M29")
   Msg_059 : BOOL ;	//FAULT NODO PROFIBUS 13 (INVERTER "M30")
   Msg_060 : BOOL ;	//FAULT NODO PROFIBUS 14 (INVERTER "M31")
   Msg_061 : BOOL ;	//FAULT NODO PROFIBUS 15 (INVERTER "M32")
   Msg_062 : BOOL ;	//FAULT NODO PROFIBUS 16 (INVERTER "M33")
   Msg_063 : BOOL ;	//FAULT NODO PROFIBUS 17 (INVERTER "M34")
   Msg_064 : BOOL ;	//FAULT NODO PROFIBUS 18 (INVERTER "M35")
   Msg_065 : BOOL ;	//FAULT NODO PROFIBUS 24 (DP/DP COUPLER FORNO)
   Msg_066 : BOOL ;	//FAULT NODO PROFIBUS 25 (ET200S - BOX JP1)
   Msg_067 : BOOL ;	//FAULT NODO PROFIBUS 26 (ET200S - BOX JP2)
   Msg_068 : BOOL ;	//FAULT NODO PROFIBUS 27 (ET200S - BOX JP3)
   Msg_069 : BOOL ;
   Msg_070 : BOOL ;	//TIMEOUT FINECORSA ALTO TRASLATORE 4 PEZZI (E20.0, E20.2)
   Msg_071 : BOOL ;	//TIMEOUT FINECORSA BASSO TRASLATORE 4 PEZZI (E20.1, E20.3)
   Msg_072 : BOOL ;	//TIMEOUT FINECORSA ALTO CATENE INGRESSO 4 PEZZI LINEA 2 (E21.4, E21.6)
   Msg_073 : BOOL ;	//TIMEOUT FINECORSA BASSO CATENE INGRESSO 4 PEZZI LINEA 2 (E21.5, E21.7)
   Msg_074 : BOOL ;	//TIMEOUT FINECORSA ALTO CATENE USCITA CADENZATORE LINEA 2 (E21.0, E21.2)
   Msg_075 : BOOL ;	//TIMEOUT FINECORSA BASSO CATENE USCITA CADENZATORE LINEA 2 (E21.1, E21.3)
   Msg_076 : BOOL ;	//TIMEOUT FINECORSA ALTO CATENE INGRESSO 4 PEZZI LINEA 1 (E22.0, E22.2)
   Msg_077 : BOOL ;	//TIMEOUT FINECORSA BASSO CATENE INGRESSO 4 PEZZI LINEA 1 (E22.1, E22.3)
   Msg_078 : BOOL ;	//TIMEOUT FINECORSA ALTO CATENE USCITA CADENZATORE LINEA 1 (E22.4, E22.6)
   Msg_079 : BOOL ;	//TIMEOUT FINECORSA BASSO CATENE USCITA CADENZATORE LINEA 1 (E22.5, E22.7)
   Msg_080 : BOOL ;	//TIMEOUT FINECORSA ALTO CATENE ACCUMULO "A" LINEA 1 (E25.0, E25.2)
   Msg_081 : BOOL ;	//TIMEOUT FINECORSA BASSO CATENE ACCUMULO "A" LINEA 1 (E25.1, E25.3)
   Msg_082 : BOOL ;	//TIMEOUT FINECORSA ALTO CATENE ACCUMULO "B" LINEA 1 (E25.4, E25.6)
   Msg_083 : BOOL ;	//TIMEOUT FINECORSA BASSO CATENE ACCUMULO "B" LINEA 1 (E25.5, E25.7)
   Msg_084 : BOOL ;	//TIMEOUT SENSORE PASSO CADENZATORE INGRESSO LINEA 2 (E24.0)
   Msg_085 : BOOL ;	//TIMEOUT SENSORE PASSO CADENZATORE INGRESSO LINEA 1 (E24.1)
   Msg_086 : BOOL ;	//TIMEOUT SENSORE PASSO CADENZATORE ACCUMULO "A" LINEA 2 (E27.2)
   Msg_087 : BOOL ;	//TIMEOUT SENSORE PASSO CADENZATORE ACCUMULO "B" LINEA 2 (E27.3)
   Msg_088 : BOOL ;
   Msg_089 : BOOL ;	//CADENZATORE INGRESSO LINEA 2 NON IN FASE (E24.0)
   Msg_090 : BOOL ;	//CADENZATORE INGRESSO LINEA 1 NON IN FASE (E24.1)
   Msg_091 : BOOL ;	//CADENZATORE ACCUMULO "A" LINEA 2 NON IN FASE (E27.2)
   Msg_092 : BOOL ;	//CADENZATORE ACCUMULO "B" LINEA 2 NON IN FASE (E27.3)
   Msg_093 : BOOL ;	//FOTOCELLULA ARRESTO PACCO 4 FILE TRASLATORE E' RIMASTA IMPEGNATA (E20.4)
   Msg_094 : BOOL ;	//FOTOCELLULA ARRESTO PACCO 4 FILE DAVANTI LINEA 2 E' RIMASTA IMPEGNATA (E23.6)
   Msg_095 : BOOL ;	//FOTOCELLULA ARRESTO PACCO 4 FILE DAVANTI LINEA 1 E' RIMASTA IMPEGNATA (E23.7)
   Msg_096 : BOOL ;	//FOTOCELLULA ARRESTO BARRA DAVANTI CADENZATORE LINEA 2 E' RIMASTA IMPEGNATA (E23
   Msg_097 : BOOL ;	//FOTOCELLULA ARRESTO BARRA DAVANTI CADENZATORE LINEA 1 E' RIMASTA IMPEGNATA (E23
   Msg_098 : BOOL ;	//FOTOCELLULA ARRESTO BARRA SU RULLIERA 1 INGRESSO ESTR. LINEA 2 E' RIMASTA IMPEG
   Msg_099 : BOOL ;	//FOTOCELLULA ARRESTO BARRA SU RULLIERA 1 INGRESSO ESTR. LINEA 1 E' RIMASTA IMPEG
   Msg_100 : BOOL ;	//FOTOCELLULA ARRESTO BARRA SU CADENZATORE ACCUMULO "A" LINEA 2 E' RIMASTA IMPEGN
   Msg_101 : BOOL ;	//FOTOCELLULA ARRESTO BARRA SU CADENZATORE ACCUMULO "B" LINEA 2 E' RIMASTA IMPEGN
   Msg_102 : BOOL ;	//FOTOCELLULA ARRESTO BARRA SU DEVIATORE ACCUMULO "A" LINEA 1 E' RIMASTA IMPEGNAT
   Msg_103 : BOOL ;	//FOTOCELLULA ARRESTO BARRA SU DEVIATORE ACCUMULO "B" LINEA 1 E' RIMASTA IMPEGNAT
   Msg_104 : BOOL ;
   Msg_105 : BOOL ;	//TIMEOUT CICLO TRASFERITORE O MANCATA LETTURA FOTOCELLULA ARRESTO CATENE (E20.4)
   Msg_106 : BOOL ;	//TIMEOUT CICLO TRASFERIMENTO 4 BARRE VERSO LINEA 2 O MANCATA LETTURA FOTOCELLULA
   Msg_107 : BOOL ;	//TIMEOUT CICLO TRASFERIMENTO 4 BARRE VERSO LINEA 1 O MANCATA LETTURA FOTOCELLULA
   Msg_108 : BOOL ;	//TIMEOUT CICLO ALIMENTAZIONE CADENZATORE LINEA 2 O MANCATA LETTURA FOTOCELLULA (
   Msg_109 : BOOL ;	//TIMEOUT CICLO ALIMENTAZIONE CADENZATORE LINEA 1 O MANCATA LETTURA FOTOCELLULA (
   Msg_110 : BOOL ;	//LINEA ACCUMULO "A" INFERIORE PIENA
   Msg_111 : BOOL ;	//LINEA ACCUMULO "A" SUPERIORE PIENA
   Msg_112 : BOOL ;	//LINEA ACCUMULO "B" INFERIORE PIENA
   Msg_113 : BOOL ;	//LINEA ACCUMULO "B" SUPERIORE PIENA
   Msg_114 : BOOL ;	//INVERTER A1 MOTORE "M20" IN ALLARME
   Msg_115 : BOOL ;	//INVERTER A2 MOTORE "M21" IN ALLARME
   Msg_116 : BOOL ;	//INVERTER A3 MOTORE "M22" IN ALLARME
   Msg_117 : BOOL ;	//INVERTER A4 MOTORE "M23" IN ALLARME
   Msg_118 : BOOL ;	//INVERTER A5 MOTORE "M24" IN ALLARME
   Msg_119 : BOOL ;	//INVERTER A6 MOTORE "M25" IN ALLARME
   Msg_120 : BOOL ;	//INVERTER A7 MOTORE "M26" IN ALLARME
   Msg_121 : BOOL ;	//INVERTER A8 MOTORE "M27" IN ALLARME
   Msg_122 : BOOL ;	//INVERTER A9 MOTORE "M28" IN ALLARME
   Msg_123 : BOOL ;	//INVERTER A10 MOTORE "M29" IN ALLARME
   Msg_124 : BOOL ;	//INVERTER A11 MOTORE "M30" IN ALLARME
   Msg_125 : BOOL ;	//INVERTER A12 MOTORE "M31" IN ALLARME
   Msg_126 : BOOL ;	//INVERTER A13 MOTORE "M32" IN ALLARME
   Msg_127 : BOOL ;	//INVERTER A14 MOTORE "M33" IN ALLARME
   Msg_128 : BOOL ;	//INVERTER A15 MOTORE "M34" IN ALLARME
   Msg_129 : BOOL ;	//INVERTER A16 MOTORE "M35" IN ALLARME
   Msg_130 : BOOL ;
   Msg_131 : BOOL ;
   Msg_132 : BOOL ;
   Msg_133 : BOOL ;
   Msg_134 : BOOL ;
   Msg_135 : BOOL ;
   Msg_136 : BOOL ;
   Msg_137 : BOOL ;
   Msg_138 : BOOL ;
   Msg_139 : BOOL ;
   Msg_140 : BOOL ;
   Msg_141 : BOOL ;
   Msg_142 : BOOL ;
   Msg_143 : BOOL ;
   Msg_144 : BOOL ;
   Msg_145 : BOOL ;
   Msg_146 : BOOL ;
   Msg_147 : BOOL ;
   Msg_148 : BOOL ;
   Msg_149 : BOOL ;
   Msg_150 : BOOL ;
   Msg_151 : BOOL ;
   Msg_152 : BOOL ;
   Msg_153 : BOOL ;
   Msg_154 : BOOL ;
   Msg_155 : BOOL ;
   Msg_156 : BOOL ;
   Msg_157 : BOOL ;
   Msg_158 : BOOL ;
   Msg_159 : BOOL ;
   Msf_160 : BOOL ;
  END_STRUCT ;
END_VAR
VAR_TEMP
  i : INT ;
  Attivo : BOOL ;
END_VAR
BEGIN
// body was compiled from an SCL source; compiled code not shown
END_FUNCTION

FUNCTION "FC_ResetAllarmi" : VOID	// FC 202
VERSION : 0.0
VAR_IN_OUT
  Allarmi : STRUCT
   Msg_001 : BOOL ;	//INTERVENTO TERMICO "KMC1" (E0.0)
   Msg_002 : BOOL ;	//INTERVENTO TERMICO "KMC2" (E0.1)
   Msg_003 : BOOL ;	//INTERVENTO TERMICO "KMC3" (E0.2)
   Msg_004 : BOOL ;	//INTERVENTO TERMICO "KMC4" (E0.3)
   Msg_005 : BOOL ;	//INTERVENTO TERMICO "KMC5" (E0.4)
   Msg_006 : BOOL ;	//INTERVENTO TERMICO "KMC6" (E0.5)
   Msg_007 : BOOL ;	//INTERVENTO TERMICO "KMC7" (E0.6)
   Msg_008 : BOOL ;	//INTERVENTO TERMICO "KMC8" (E0.7)
   Msg_009 : BOOL ;	//INTERVENTO TERMICO "KMC9" (E1.0)
   Msg_010 : BOOL ;	//INTERVENTO TERMICO "KMC10" (E1.1)
   Msg_011 : BOOL ;	//INTERVENTO TERMICO "KMC11" (E1.2)
   Msg_012 : BOOL ;	//INTERVENTO TERMICO "KMC12" (E1.3)
   Msg_013 : BOOL ;	//INTERVENTO TERMICO "KMC13" (E1.4)
   Msg_014 : BOOL ;	//INTERVENTO TERMICO "KMC14" (E1.5)
   Msg_015 : BOOL ;	//INTERVENTO TERMICO "KMC15" (E1.6)
   Msg_016 : BOOL ;	//INTERVENTO TERMICO "KMC16" (E1.7)
   Msg_017 : BOOL ;	//INTERVENTO TERMICO "KMC17" (E2.0)
   Msg_018 : BOOL ;	//INTERVENTO TERMICO "KMC18" (E2.1)
   Msg_019 : BOOL ;	//INTERVENTO TERMICO "KMC19" (E2.2)
   Msg_020 : BOOL ;	//INTERVENTO TERMICO "KMC20" (E2.3)
   Msg_021 : BOOL ;	//INTERVENTO TERMICO "QF20" ALIM. INVERTER A1 "M20" (E3.0)
   Msg_022 : BOOL ;	//INTERVENTO TERMICO "QF21" ALIM. INVERTER A2 "M21" (E3.1)
   Msg_023 : BOOL ;	//INTERVENTO TERMICO "QF22" ALIM. INVERTER A3 "M22" (E3.2)
   Msg_024 : BOOL ;	//INTERVENTO TERMICO "QF23" ALIM. INVERTER A4 "M23" (E3.3)
   Msg_025 : BOOL ;	//INTERVENTO TERMICO "QF24" ALIM. INVERTER A5 "M24" (E3.4)
   Msg_026 : BOOL ;	//INTERVENTO TERMICO "QF25" ALIM. INVERTER A6 "M25" (E3.5)
   Msg_027 : BOOL ;	//INTERVENTO TERMICO "QF26" ALIM. INVERTER A7 "M26" (E3.6)
   Msg_028 : BOOL ;	//INTERVENTO TERMICO "QF27" ALIM. INVERTER A8 "M27" (E3.7)
   Msg_029 : BOOL ;	//INTERVENTO TERMICO "QF28" ALIM. INVERTER A9 "M28" (E4.0)
   Msg_030 : BOOL ;	//INTERVENTO TERMICO "QF29" ALIM. INVERTER A10 "M29" (E4.1)
   Msg_031 : BOOL ;	//INTERVENTO TERMICO "QF30" ALIM. INVERTER A11 "M30" (E4.2)
   Msg_032 : BOOL ;	//INTERVENTO TERMICO "QF31" ALIM. INVERTER A12 "M31" (E4.3)
   Msg_033 : BOOL ;	//INTERVENTO TERMICO "QF32" ALIM. INVERTER A13 "M32" (E4.4)
   Msg_034 : BOOL ;	//INTERVENTO TERMICO "QF33" ALIM. INVERTER A14 "M33" (E4.5)
   Msg_035 : BOOL ;	//INTERVENTO TERMICO "QF34" ALIM. INVERTER A15 "M34" (E4.6)
   Msg_036 : BOOL ;	//INTERVENTO TERMICO "QF35" ALIM. INVERTER A16 "M35" (E4.7)
   Msg_037 : BOOL ;	//INTERVENTO TERMICO "QF36"(E5.0)
   Msg_038 : BOOL ;
   Msg_039 : BOOL ;
   Msg_040 : BOOL ;
   Msg_041 : BOOL ;	//INTERVENTO PROTEZIONE "QF6" VENTILAZIONE QUADRO (E5.1)
   Msg_042 : BOOL ;	//INTERVENTO PROTEZIONE "QF8"  (E5.2)
   Msg_043 : BOOL ;	//INTERVENTO PROTEZIONE "QF19" ALIM. CIRCUITI D'EMERGENZA  (E5.3)
   Msg_044 : BOOL ;	//INTERVENTO PROTEZIONE "QF10" ALIM. COMANDI QUADRO (E5.4)
   Msg_045 : BOOL ;	//INTERVENTO PROTEZIONE "QF11" ALIM. COMANDI JP1  (E5.5)
   Msg_046 : BOOL ;	//INTERVENTO PROTEZIONE "QF12" ALIM. COMANDI JP2  (E5.6)
   Msg_047 : BOOL ;	//INTERVENTO PROTEZIONE "QF13" ALIM. COMANDI JP3  (E5.7)
   Msg_048 : BOOL ;
   Msg_049 : BOOL ;	//FAULT NODO PROFIBUS 3 (INVERTER "M20")
   Msg_050 : BOOL ;	//FAULT NODO PROFIBUS 4 (INVERTER "M21")
   Msg_051 : BOOL ;	//FAULT NODO PROFIBUS 5 (INVERTER "M22")
   Msg_052 : BOOL ;	//FAULT NODO PROFIBUS 6 (INVERTER "M23")
   Msg_053 : BOOL ;	//FAULT NODO PROFIBUS 7 (INVERTER "M24")
   Msg_054 : BOOL ;	//FAULT NODO PROFIBUS 8 (INVERTER "M25")
   Msg_055 : BOOL ;	//FAULT NODO PROFIBUS 9 (INVERTER "M26")
   Msg_056 : BOOL ;	//FAULT NODO PROFIBUS 10 (INVERTER "M27")
   Msg_057 : BOOL ;	//FAULT NODO PROFIBUS 11 (INVERTER "M28")
   Msg_058 : BOOL ;	//FAULT NODO PROFIBUS 12 (INVERTER "M29")
   Msg_059 : BOOL ;	//FAULT NODO PROFIBUS 13 (INVERTER "M30")
   Msg_060 : BOOL ;	//FAULT NODO PROFIBUS 14 (INVERTER "M31")
   Msg_061 : BOOL ;	//FAULT NODO PROFIBUS 15 (INVERTER "M32")
   Msg_062 : BOOL ;	//FAULT NODO PROFIBUS 16 (INVERTER "M33")
   Msg_063 : BOOL ;	//FAULT NODO PROFIBUS 17 (INVERTER "M34")
   Msg_064 : BOOL ;	//FAULT NODO PROFIBUS 18 (INVERTER "M35")
   Msg_065 : BOOL ;	//FAULT NODO PROFIBUS 24 (DP/DP COUPLER FORNO)
   Msg_066 : BOOL ;	//FAULT NODO PROFIBUS 25 (ET200S - BOX JP1)
   Msg_067 : BOOL ;	//FAULT NODO PROFIBUS 26 (ET200S - BOX JP2)
   Msg_068 : BOOL ;	//FAULT NODO PROFIBUS 27 (ET200S - BOX JP3)
   Msg_069 : BOOL ;
   Msg_070 : BOOL ;	//TIMEOUT FINECORSA ALTO TRASLATORE 4 PEZZI (E20.0, E20.2)
   Msg_071 : BOOL ;	//TIMEOUT FINECORSA BASSO TRASLATORE 4 PEZZI (E20.1, E20.3)
   Msg_072 : BOOL ;	//TIMEOUT FINECORSA ALTO CATENE INGRESSO 4 PEZZI LINEA 2 (E21.4, E21.6)
   Msg_073 : BOOL ;	//TIMEOUT FINECORSA BASSO CATENE INGRESSO 4 PEZZI LINEA 2 (E21.5, E21.7)
   Msg_074 : BOOL ;	//TIMEOUT FINECORSA ALTO CATENE USCITA CADENZATORE LINEA 2 (E21.0, E21.2)
   Msg_075 : BOOL ;	//TIMEOUT FINECORSA BASSO CATENE USCITA CADENZATORE LINEA 2 (E21.1, E21.3)
   Msg_076 : BOOL ;	//TIMEOUT FINECORSA ALTO CATENE INGRESSO 4 PEZZI LINEA 1 (E22.0, E22.2)
   Msg_077 : BOOL ;	//TIMEOUT FINECORSA BASSO CATENE INGRESSO 4 PEZZI LINEA 1 (E22.1, E22.3)
   Msg_078 : BOOL ;	//TIMEOUT FINECORSA ALTO CATENE USCITA CADENZATORE LINEA 1 (E22.4, E22.6)
   Msg_079 : BOOL ;	//TIMEOUT FINECORSA BASSO CATENE USCITA CADENZATORE LINEA 1 (E22.5, E22.7)
   Msg_080 : BOOL ;	//TIMEOUT FINECORSA ALTO CATENE ACCUMULO "A" LINEA 1 (E25.0, E25.2)
   Msg_081 : BOOL ;	//TIMEOUT FINECORSA BASSO CATENE ACCUMULO "A" LINEA 1 (E25.1, E25.3)
   Msg_082 : BOOL ;	//TIMEOUT FINECORSA ALTO CATENE ACCUMULO "B" LINEA 1 (E25.4, E25.6)
   Msg_083 : BOOL ;	//TIMEOUT FINECORSA BASSO CATENE ACCUMULO "B" LINEA 1 (E25.5, E25.7)
   Msg_084 : BOOL ;	//TIMEOUT SENSORE PASSO CADENZATORE INGRESSO LINEA 2 (E24.0)
   Msg_085 : BOOL ;	//TIMEOUT SENSORE PASSO CADENZATORE INGRESSO LINEA 1 (E24.1)
   Msg_086 : BOOL ;	//TIMEOUT SENSORE PASSO CADENZATORE ACCUMULO "A" LINEA 2 (E27.2)
   Msg_087 : BOOL ;	//TIMEOUT SENSORE PASSO CADENZATORE ACCUMULO "B" LINEA 2 (E27.3)
   Msg_088 : BOOL ;
   Msg_089 : BOOL ;	//CADENZATORE INGRESSO LINEA 2 NON IN FASE (E24.0)
   Msg_090 : BOOL ;	//CADENZATORE INGRESSO LINEA 1 NON IN FASE (E24.1)
   Msg_091 : BOOL ;	//CADENZATORE ACCUMULO "A" LINEA 2 NON IN FASE (E27.2)
   Msg_092 : BOOL ;	//CADENZATORE ACCUMULO "B" LINEA 2 NON IN FASE (E27.3)
   Msg_093 : BOOL ;	//FOTOCELLULA ARRESTO PACCO 4 FILE TRASLATORE E' RIMASTA IMPEGNATA (E20.4)
   Msg_094 : BOOL ;	//FOTOCELLULA ARRESTO PACCO 4 FILE DAVANTI LINEA 2 E' RIMASTA IMPEGNATA (E23.6)
   Msg_095 : BOOL ;	//FOTOCELLULA ARRESTO PACCO 4 FILE DAVANTI LINEA 1 E' RIMASTA IMPEGNATA (E23.7)
   Msg_096 : BOOL ;	//FOTOCELLULA ARRESTO BARRA DAVANTI CADENZATORE LINEA 2 E' RIMASTA IMPEGNATA (E23
   Msg_097 : BOOL ;	//FOTOCELLULA ARRESTO BARRA DAVANTI CADENZATORE LINEA 1 E' RIMASTA IMPEGNATA (E23
   Msg_098 : BOOL ;	//FOTOCELLULA ARRESTO BARRA SU RULLIERA 1 INGRESSO ESTR. LINEA 2 E' RIMASTA IMPEG
   Msg_099 : BOOL ;	//FOTOCELLULA ARRESTO BARRA SU RULLIERA 1 INGRESSO ESTR. LINEA 1 E' RIMASTA IMPEG
   Msg_100 : BOOL ;	//FOTOCELLULA ARRESTO BARRA SU CADENZATORE ACCUMULO "A" LINEA 2 E' RIMASTA IMPEGN
   Msg_101 : BOOL ;	//FOTOCELLULA ARRESTO BARRA SU CADENZATORE ACCUMULO "B" LINEA 2 E' RIMASTA IMPEGN
   Msg_102 : BOOL ;	//FOTOCELLULA ARRESTO BARRA SU DEVIATORE ACCUMULO "A" LINEA 1 E' RIMASTA IMPEGNAT
   Msg_103 : BOOL ;	//FOTOCELLULA ARRESTO BARRA SU DEVIATORE ACCUMULO "B" LINEA 1 E' RIMASTA IMPEGNAT
   Msg_104 : BOOL ;
   Msg_105 : BOOL ;	//TIMEOUT CICLO TRASFERITORE O MANCATA LETTURA FOTOCELLULA ARRESTO CATENE (E20.4)
   Msg_106 : BOOL ;	//TIMEOUT CICLO TRASFERIMENTO 4 BARRE VERSO LINEA 2 O MANCATA LETTURA FOTOCELLULA
   Msg_107 : BOOL ;	//TIMEOUT CICLO TRASFERIMENTO 4 BARRE VERSO LINEA 1 O MANCATA LETTURA FOTOCELLULA
   Msg_108 : BOOL ;	//TIMEOUT CICLO ALIMENTAZIONE CADENZATORE LINEA 2 O MANCATA LETTURA FOTOCELLULA (
   Msg_109 : BOOL ;	//TIMEOUT CICLO ALIMENTAZIONE CADENZATORE LINEA 1 O MANCATA LETTURA FOTOCELLULA (
   Msg_110 : BOOL ;	//LINEA ACCUMULO "A" INFERIORE PIENA
   Msg_111 : BOOL ;	//LINEA ACCUMULO "A" SUPERIORE PIENA
   Msg_112 : BOOL ;	//LINEA ACCUMULO "B" INFERIORE PIENA
   Msg_113 : BOOL ;	//LINEA ACCUMULO "B" SUPERIORE PIENA
   Msg_114 : BOOL ;	//INVERTER A1 MOTORE "M20" IN ALLARME
   Msg_115 : BOOL ;	//INVERTER A2 MOTORE "M21" IN ALLARME
   Msg_116 : BOOL ;	//INVERTER A3 MOTORE "M22" IN ALLARME
   Msg_117 : BOOL ;	//INVERTER A4 MOTORE "M23" IN ALLARME
   Msg_118 : BOOL ;	//INVERTER A5 MOTORE "M24" IN ALLARME
   Msg_119 : BOOL ;	//INVERTER A6 MOTORE "M25" IN ALLARME
   Msg_120 : BOOL ;	//INVERTER A7 MOTORE "M26" IN ALLARME
   Msg_121 : BOOL ;	//INVERTER A8 MOTORE "M27" IN ALLARME
   Msg_122 : BOOL ;	//INVERTER A9 MOTORE "M28" IN ALLARME
   Msg_123 : BOOL ;	//INVERTER A10 MOTORE "M29" IN ALLARME
   Msg_124 : BOOL ;	//INVERTER A11 MOTORE "M30" IN ALLARME
   Msg_125 : BOOL ;	//INVERTER A12 MOTORE "M31" IN ALLARME
   Msg_126 : BOOL ;	//INVERTER A13 MOTORE "M32" IN ALLARME
   Msg_127 : BOOL ;	//INVERTER A14 MOTORE "M33" IN ALLARME
   Msg_128 : BOOL ;	//INVERTER A15 MOTORE "M34" IN ALLARME
   Msg_129 : BOOL ;	//INVERTER A16 MOTORE "M35" IN ALLARME
   Msg_130 : BOOL ;
   Msg_131 : BOOL ;
   Msg_132 : BOOL ;
   Msg_133 : BOOL ;
   Msg_134 : BOOL ;
   Msg_135 : BOOL ;
   Msg_136 : BOOL ;
   Msg_137 : BOOL ;
   Msg_138 : BOOL ;
   Msg_139 : BOOL ;
   Msg_140 : BOOL ;
   Msg_141 : BOOL ;
   Msg_142 : BOOL ;
   Msg_143 : BOOL ;
   Msg_144 : BOOL ;
   Msg_145 : BOOL ;
   Msg_146 : BOOL ;
   Msg_147 : BOOL ;
   Msg_148 : BOOL ;
   Msg_149 : BOOL ;
   Msg_150 : BOOL ;
   Msg_151 : BOOL ;
   Msg_152 : BOOL ;
   Msg_153 : BOOL ;
   Msg_154 : BOOL ;
   Msg_155 : BOOL ;
   Msg_156 : BOOL ;
   Msg_157 : BOOL ;
   Msg_158 : BOOL ;
   Msg_159 : BOOL ;
   Msf_160 : BOOL ;
  END_STRUCT ;
END_VAR
VAR_TEMP
  i : INT ;
END_VAR
BEGIN
// body was compiled from an SCL source; compiled code not shown
END_FUNCTION

FUNCTION "FC_ControlloMsgEth" : VOID	// FC 203
VERSION : 0.0
VAR_INPUT
  Str : STRING  [254 ];
END_VAR
VAR_OUTPUT
  MsgL1 : BOOL ;	//La stringa Str inizia con "L1"
  MsgL2 : BOOL ;	//La stringa Str inizia con "L2"
END_VAR
VAR_TEMP
  N : INT ;
  Ch : CHAR ;
END_VAR
BEGIN
// body was compiled from an SCL source; compiled code not shown
END_FUNCTION

FUNCTION "InvertiMinuscMaiusc" : VOID	// FC 204
VERSION : 0.0
VAR_INPUT
  StrIn : STRING  [254 ];
END_VAR
VAR_OUTPUT
  StrOut : STRING  [254 ];
END_VAR
VAR_TEMP
  I : INT ;
  N : INT ;
  Ch : CHAR ;
END_VAR
BEGIN
// body was compiled from an SCL source; compiled code not shown
END_FUNCTION

DATA_BLOCK "DB_OP"	// DB 2
//
// Commento al blocco ...
//
//
VERSION : 0.0
  STRUCT
   PaginaRichiesta : INT ;	//Pagina richiesta sul pannello
   CambiaPagina : INT ;	//La modifica di questo valore forza il cambio pagina sul pannello
   Aux : ARRAY  [1 .. 10 ] OF DINT ;
   InfoPagina : STRUCT
    TipoPagina : WORD ;
    PaginaCorrente : INT ;
    Riservato1 : INT ;
    CampoCorrente : INT ;
    Riservato2 : INT ;
   END_STRUCT ;
   TastiGenerici : STRUCT
    Tasto_1 : BOOL ;
    Tasto_2 : BOOL ;
    Tasto_3 : BOOL ;
    Tasto_4 : BOOL ;
    Tasto_5 : BOOL ;
    Tasto_6 : BOOL ;
    Tasto_7 : BOOL ;
    Tasto_8 : BOOL ;
    Tasto_9 : BOOL ;
    Tasto_10 : BOOL ;
    Tasto_11 : BOOL ;
    Tasto_12 : BOOL ;
    Tasto_13 : BOOL ;
    Tasto_14 : BOOL ;
    Tasto_15 : BOOL ;
    Tasto_16 : BOOL ;
   END_STRUCT ;
   Allarmi : UDT 101;	//Messaggi di allarme su
   Segnalazioni : UDT 102;	//Segnalazioni su pannello
   Manuali : UDT 100;	//Comandi manuali da pannello
   StatoImpianto : INT ;	//0: --; 1: MANUALE; 2: AUTOMATICO
   dummy : ARRAY  [1 .. 49 ] OF INT ;
   MsgEthPort2000 : STRING  [64 ];	//Stringa ricevuta dal termiale linea 1
   MsgEthPort2001 : STRING  [64 ];	//Stringa ricevuta dal termiale linea 2
  END_STRUCT ;	
BEGIN
END_DATA_BLOCK

DATA_BLOCK "DB_InverterParams"	// DB 3
//
// Parametri inverter
//
//
VERSION : 0.0
  STRUCT
   Params : ARRAY  [20 .. 35 ] OF UDT 202;
  END_STRUCT ;	
BEGIN
END_DATA_BLOCK

DATA_BLOCK "DETAIL_DIAG_DB"	// DB 125
VERSION : 0.0
"DETAIL_DP_DIAG"
BEGIN
END_DATA_BLOCK

DATA_BLOCK "DB_ReadParamLoop"	// DB 211
VERSION : 0.0
"FB_ReadParamLoop"
BEGIN
END_DATA_BLOCK

DATA_BLOCK "DB_GestCodeEstrusori"	// DB 212
VERSION : 0.0
"FB_GestCodeEstrusori"
BEGIN
END_DATA_BLOCK

DATA_BLOCK "DB_LinkEthernet_1"	// DB 213
AUTHOR : Filip1
FAMILY : Ethernet
VERSION : 0.0
"FB_LinkEthernet"
BEGIN
END_DATA_BLOCK

DATA_BLOCK "DB_LinkEthernet_2"	// DB 214
AUTHOR : Filip1
FAMILY : Ethernet
VERSION : 0.0
"FB_LinkEthernet"
BEGIN
END_DATA_BLOCK

ORGANIZATION_BLOCK OB 1
TITLE = "Main Program Sweep (Cycle)"
VERSION : 0.1
VAR_TEMP
  OB1_EV_CLASS : BYTE ;	//Bits 0-3 = 1 (Coming event), Bits 4-7 = 1 (Event class 1)
  OB1_SCAN_1 : BYTE ;	//1 (Cold restart scan 1 of OB 1), 3 (Scan 2-n of OB 1)
  OB1_PRIORITY : BYTE ;	//Priority of OB Execution
  OB1_OB_NUMBR : BYTE ;	//1 (Organization block 1, OB1)
  OB1_RESERVED_1 : BYTE ;	//Reserved for system
  OB1_RESERVED_2 : BYTE ;	//Reserved for system
  OB1_PREV_CYCLE : INT ;	//Cycle time of previous OB1 scan (milliseconds)
  OB1_MIN_CYCLE : INT ;	//Minimum cycle time of OB1 (milliseconds)
  OB1_MAX_CYCLE : INT ;	//Maximum cycle time of OB1 (milliseconds)
  OB1_DATE_TIME : DATE_AND_TIME ;	//Date and time OB1 started
END_VAR
BEGIN
NETWORK
TITLE = GENERAZIONE BIT AUSILIARI
      SET;
      R     "OFF";
      S     "ON";
      R     "TODO";
      S     "BYPASS";
      L     "ClockBits";
      L     "MemClockBits";
      XOW;
      L     "ClockBits";
      T     "MemClockBits";
      AW;
      T     "ImpClockBits";
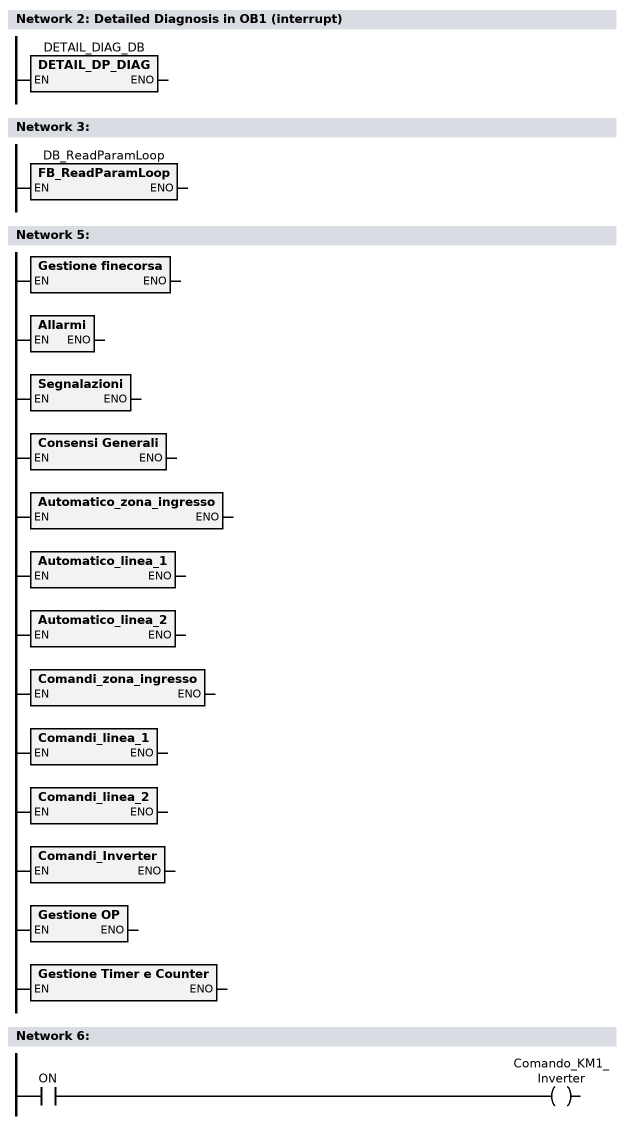
NETWORK
TITLE = Detailed Diagnosis in OB1 (interrupt)
      CALL  "DETAIL_DP_DIAG" , "DETAIL_DIAG_DB";
NETWORK
TITLE =
      CALL  "FB_ReadParamLoop" , "DB_ReadParamLoop";
NETWORK
TITLE =
// (network holds code this reader does not know; not shown)
//Se ricecuta nuova stringa da ethernt
//verifico se ricevuto L1 o L2 e accordo
//Se ricecuta nuova stringa da ethernt
//verifico se ricevuto L1 o L2 e accordo
NETWORK
TITLE =
      CALL  "Gestione finecorsa";
      CALL  "Allarmi";
      CALL  "Segnalazioni";
      CALL  "Consensi Generali";
      CALL  "Automatico_zona_ingresso";
      CALL  "Automatico_linea_1";
      CALL  "Automatico_linea_2";
      CALL  "Comandi_zona_ingresso";
      CALL  "Comandi_linea_1";
      CALL  "Comandi_linea_2";
      CALL  "Comandi_Inverter";
      CALL  "Gestione OP";
      CALL  "Gestione Timer e Counter";
NETWORK
TITLE =
      A     "ON";
      =     "Comando_KM1_Inverter";
NETWORK
TITLE =
      BE;
END_ORGANIZATION_BLOCK

ORGANIZATION_BLOCK "CYCL_FLT"	// OB 80
TITLE = "Cycle Time Fault"
AUTHOR : PROTEKNO
VERSION : 0.1
VAR_TEMP
  OB80_EV_CLASS : BYTE ;	//16#35, Event class 3, Entering event state, Internal fault event
  OB80_FLT_ID : BYTE ;	//16#XX, Fault identifcation code
  OB80_PRIORITY : BYTE ;	//Priority of OB Execution
  OB80_OB_NUMBR : BYTE ;	//80 (Organization block 80, OB80)
  OB80_RESERVED_1 : BYTE ;	//Reserved for system
  OB80_RESERVED_2 : BYTE ;	//Reserved for system
  OB80_ERROR_INFO : WORD ;	//Error information on event
  OB80_ERR_EV_CLASS : BYTE ;	//Class of event causing error
  OB80_ERR_EV_NUM : BYTE ;	//Number of event causing error
  OB80_OB_PRIORITY : BYTE ;	//Priority of OB causing error
  OB80_OB_NUM : BYTE ;	//Number of OB causing error
  OB80_DATE_TIME : DATE_AND_TIME ;	//Date and time OB80 started
END_VAR
BEGIN
// (block stored without names or comments; labels and parameter names are numbered)
END_ORGANIZATION_BLOCK

ORGANIZATION_BLOCK "I/O_FLT1"	// OB 82
TITLE = "I/O Point Fault"
AUTHOR : PROTEKNO
VERSION : 0.1
VAR_TEMP
  OB82_EV_CLASS : BYTE ;	//16#39, Event class 3, Entering event state, Internal fault event
  OB82_FLT_ID : BYTE ;	//16#XX, Fault identifcation code
  OB82_PRIORITY : BYTE ;	//Priority of OB Execution
  OB82_OB_NUMBR : BYTE ;	//82 (Organization block 82, OB82)
  OB82_RESERVED_1 : BYTE ;	//Reserved for system
  OB82_IO_FLAG : BYTE ;	//Input (01010100), Output (01010101)
  OB82_MDL_ADDR : WORD ;	//Base address of module with fault
  OB82_MDL_DEFECT : BOOL ;	//Module defective
  OB82_INT_FAULT : BOOL ;	//Internal fault
  OB82_EXT_FAULT : BOOL ;	//External fault
  OB82_PNT_INFO : BOOL ;	//Point information
  OB82_EXT_VOLTAGE : BOOL ;	//External voltage low
  OB82_FLD_CONNCTR : BOOL ;	//Field wiring connector missing
  OB82_NO_CONFIG : BOOL ;	//Module has no configuration data
  OB82_CONFIG_ERR : BOOL ;	//Module has configuration error
  OB82_MDL_TYPE : BYTE ;	//Type of module
  OB82_SUB_MDL_ERR : BOOL ;	//Sub-Module is missing or has error
  OB82_COMM_FAULT : BOOL ;	//Communication fault
  OB82_MDL_STOP : BOOL ;	//Module is stopped
  OB82_WTCH_DOG_FLT : BOOL ;	//Watch dog timer stopped module
  OB82_INT_PS_FLT : BOOL ;	//Internal power supply fault
  OB82_PRIM_BATT_FLT : BOOL ;	//Primary battery is in fault
  OB82_BCKUP_BATT_FLT : BOOL ;	//Backup battery is in fault
  OB82_RESERVED_2 : BOOL ;	//Reserved for system
  OB82_RACK_FLT : BOOL ;	//Rack fault, only for bus interface module
  OB82_PROC_FLT : BOOL ;	//Processor fault
  OB82_EPROM_FLT : BOOL ;	//EPROM fault
  OB82_RAM_FLT : BOOL ;	//RAM fault
  OB82_ADU_FLT : BOOL ;	//ADU fault
  OB82_FUSE_FLT : BOOL ;	//Fuse fault
  OB82_HW_INTR_FLT : BOOL ;	//Hardware interupt input in fault
  OB82_RESERVED_3 : BOOL ;	//Reserved for system
  OB82_DATE_TIME : DATE_AND_TIME ;	//Date and time OB82 started
END_VAR
BEGIN
NETWORK
TITLE =
      CALL  "DETAIL_DP_DIAG" , "DETAIL_DIAG_DB";
END_ORGANIZATION_BLOCK

